KUKA KRL program: MyProgram_241().src

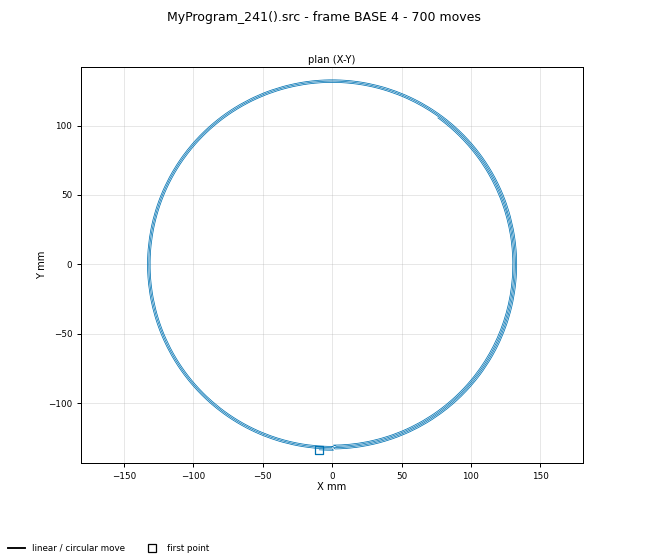
[picture p0: tool path of MyProgram_241().src in frame BASE 4, 700 of 700 moves have a stored position in this frame; points joined in program order, loops and branches not executed]
&ACCESS RVP
&REL 1
&PARAM TEMPLATE = C:\KRC\Roboter\Template\vorgabe
&PARAM EDITMASK = *
DEF MyProgram_241()
; ---- Setting reference (Base) ----
$BASE = BASE_DATA[4]

; --------------------------
; ---- Setting tool (TCP) ----
$TOOL = TOOL_DATA[3]
; --------------------------

$VEL.CP = VEL_APROX_PRINT
Startdeposition()
$VEL.CP = VEL_PRINT
LIN {X -9.2495,Y -133.5203,Z 161,A -94.9072,B 19.4805,C -0.419,E1 19.4752,E2 543.1799} C_DIS
LIN {X -6.5634,Y -133.6784,Z 161,A -93.7655,B 19.4805,C -0.4187,E1 19.4784,E2 542.039} C_DIS
LIN {X -3.4511,Y -133.7952,Z 161,A -92.3278,B 19.4805,C -0.4231,E1 19.4824,E2 540.5877} C_DIS
LIN {X 0.9612,Y -133.8342,Z 161,A -90.53,B 19.4805,C -0.4197,E1 19.4874,E2 538.8002} C_DIS
Enddeposition()
LIN {X 0.9612,Y -133.8342,Z 161,A -90.53,B 19.4805,C -0.4197,E1 19.4874,E2 538.8002} C_DIS
Startdeposition()
$VEL.CP = VEL_PRINT
LIN {X 0.1384,Y -132.9165,Z 161,A -91.2361,B 18.2986,C -0.2589,E1 18.2997,E2 539.9083} C_DIS
LIN {X -4.1167,Y -132.8521,Z 161,A -93.0475,B 18.2986,C -0.2596,E1 18.2947,E2 541.7178} C_DIS
LIN {X -8.2426,Y -132.6594,Z 161,A -94.8169,B 18.2986,C -0.26,E1 18.2897,E2 543.4865} C_DIS
LIN {X -12.4116,Y -132.3347,Z 161,A -96.6477,B 18.2986,C -0.2591,E1 18.2846,E2 545.3213} C_DIS
LIN {X -16.3847,Y -131.9029,Z 161,A -98.3665,B 18.2986,C -0.2596,E1 18.2799,E2 547.0403} C_DIS
LIN {X -20.2854,Y -131.3579,Z 161,A -99.987,B 18.2986,C -0.263,E1 18.2754,E2 548.6519} C_DIS
LIN {X -24.0292,Y -130.7264,Z 161,A -101.7483,B 18.2986,C -0.2589,E1 18.2705,E2 550.4286} C_DIS
LIN {X -28.0957,Y -129.9116,Z 161,A -103.4109,B 18.2986,C -0.2644,E1 18.266,E2 552.0765} C_DIS
LIN {X -35.5368,Y -128.0764,Z 161,A -106.7188,B 18.2985,C -0.2661,E1 18.2571,E2 555.3853} C_DIS
LIN {X -38.6101,Y -127.1837,Z 161,A -107.9788,B 18.2984,C -0.2716,E1 18.2537,E2 556.6309} C_DIS
LIN {X -43.386,Y -125.6345,Z 161,A -110.1035,B 18.2984,C -0.2748,E1 18.2481,E2 558.7509} C_DIS
LIN {X -46.3353,Y -124.5771,Z 161,A -111.6534,B 18.2984,C -0.2686,E1 18.244,E2 560.3249} C_DIS
LIN {X -49.0204,Y -123.547,Z 161,A -112.8623,B 18.2984,C -0.2709,E1 18.2408,E2 561.5301} C_DIS
LIN {X -52.3507,Y -122.1716,Z 161,A -114.4846,B 18.2984,C -0.27,E1 18.2366,E2 563.1605} C_DIS
LIN {X -55.4455,Y -120.7984,Z 161,A -115.9124,B 18.2984,C -0.2728,E1 18.233,E2 564.5843} C_DIS
LIN {X -58.5683,Y -119.3152,Z 161,A -117.3737,B 18.2984,C -0.2756,E1 18.2294,E2 566.0418} C_DIS
LIN {X -61.6117,Y -117.7724,Z 161,A -118.8799,B 18.2984,C -0.2762,E1 18.2256,E2 567.5519} C_DIS
LIN {X -65.3546,Y -115.7397,Z 161,A -120.716,B 18.2983,C -0.2786,E1 18.2211,E2 569.3877} C_DIS
LIN {X -68.6279,Y -113.8291,Z 161,A -122.4205,B 18.2983,C -0.2784,E1 18.217,E2 571.1001} C_DIS
LIN {X -72.315,Y -111.523,Z 161,A -124.324,B 18.2983,C -0.2802,E1 18.2125,E2 573.0064} C_DIS
LIN {X -75.3253,Y -109.5123,Z 161,A -126.0329,B 18.2983,C -0.2774,E1 18.2085,E2 574.7324} C_DIS
LIN {X -78.2414,Y -107.4486,Z 161,A -127.5386,B 18.2983,C -0.2812,E1 18.2051,E2 576.2334} C_DIS
LIN {X -82.235,Y -104.4235,Z 161,A -129.4084,B 18.298,C -0.2954,E1 18.2011,E2 578.0674} C_DIS
LIN {X -86.685,Y -100.7598,Z 161,A -132.0769,B 18.298,C -0.2934,E1 18.1953,E2 580.7566} C_DIS
LIN {X -90.3322,Y -97.504,Z 161,A -134.3348,B 18.298,C -0.2922,E1 18.1906,E2 583.0312} C_DIS
LIN {X -93.9479,Y -94.0253,Z 161,A -136.4373,B 18.298,C -0.2987,E1 18.1864,E2 585.1252} C_DIS
LIN {X -97.0592,Y -90.8099,Z 161,A -138.3595,B 18.298,C -0.3031,E1 18.1827,E2 587.0452} C_DIS
LIN {X -101.3952,Y -85.9412,Z 161,A -141.1571,B 18.2978,C -0.3098,E1 18.1776,E2 589.8391} C_DIS
LIN {X -103.6083,Y -83.2598,Z 161,A -142.773,B 18.2978,C -0.3091,E1 18.1747,E2 591.4678} C_DIS
LIN {X -106.4807,Y -79.5533,Z 161,A -144.7225,B 18.2978,C -0.3164,E1 18.1714,E2 593.407} C_DIS
LIN {X -109.0968,Y -75.9258,Z 161,A -146.6648,B 18.2976,C -0.3206,E1 18.1683,E2 595.3493} C_DIS
LIN {X -110.9412,Y -73.2045,Z 161,A -147.9595,B 18.2975,C -0.3284,E1 18.1663,E2 596.628} C_DIS
LIN {X -113.1832,Y -69.6881,Z 161,A -149.914,B 18.2975,C -0.3275,E1 18.1634,E2 598.5995} C_DIS
LIN {X -115.5866,Y -65.625,Z 161,A -151.9354,B 18.2975,C -0.3332,E1 18.1606,E2 600.6173} C_DIS
LIN {X -117.4844,Y -62.1602,Z 161,A -153.6006,B 18.2973,C -0.3391,E1 18.1584,E2 602.2761} C_DIS
LIN {X -118.8433,Y -59.525,Z 161,A -155.4953,B 18.2976,C -0.3212,E1 18.1559,E2 604.2426} C_DIS
LIN {X -120.9937,Y -55.0223,Z 161,A -157.1772,B 18.2972,C -0.3432,E1 18.154,E2 605.8667} C_DIS
LIN {X -122.5718,Y -51.4053,Z 161,A -158.7371,B 18.2971,C -0.3529,E1 18.1523,E2 607.4078} C_DIS
LIN {X -124.1426,Y -47.4915,Z 161,A -160.6737,B 18.2971,C -0.3539,E1 18.1503,E2 609.3565} C_DIS
LIN {X -125.4984,Y -43.7786,Z 161,A -162.2899,B 18.2969,C -0.3618,E1 18.1488,E2 610.9603} C_DIS
LIN {X -126.4864,Y -40.8374,Z 161,A -163.639,B 18.2969,C -0.3653,E1 18.1476,E2 612.3091} C_DIS
LIN {X -127.5295,Y -37.4513,Z 161,A -165.1262,B 18.2967,C -0.3712,E1 18.1464,E2 613.7896} C_DIS
LIN {X -128.4618,Y -34.1165,Z 161,A -166.6183,B 18.2967,C -0.3756,E1 18.1453,E2 615.2798} C_DIS
LIN {X -129.2371,Y -31.0509,Z 161,A -168.1072,B 18.2967,C -0.3753,E1 18.1443,E2 616.7819} C_DIS
LIN {X -130.3279,Y -26.0999,Z 161,A -170.7821,B 18.2968,C -0.3652,E1 18.1428,E2 619.5116} C_DIS
LIN {X -131.1102,Y -21.829,Z 161,A -172.1204,B 18.2964,C -0.389,E1 18.1422,E2 620.7845} C_DIS
LIN {X -132.1507,Y -14.2347,Z 161,A -175.3713,B 18.2961,C -0.4009,E1 18.141,E2 624.0247} C_DIS
LIN {X -132.5626,Y -9.6743,Z 161,A -177.4773,B 18.2961,C -0.4024,E1 18.1405,E2 626.1437} C_DIS
LIN {X -132.7947,Y -5.6803,Z 161,A -179.2819,B 18.2961,C -0.405,E1 18.1402,E2 627.9553} C_DIS
LIN {X -132.8975,Y -2.1736,Z 161,A 179.0637,B 18.2961,C -0.4049,E1 18.1402,E2 629.6243} C_DIS
LIN {X -132.8525,Y 4.1024,Z 161,A 176.4408,B 18.2958,C -0.4161,E1 18.1402,E2 632.2336} C_DIS
LIN {X -132.6983,Y 7.6106,Z 161,A 175.0478,B 18.2956,C -0.4249,E1 18.1405,E2 633.6102} C_DIS
LIN {X -132.4708,Y 10.8636,Z 161,A 173.4125,B 18.2956,C -0.4214,E1 18.1408,E2 635.2704} C_DIS
LIN {X -131.5776,Y 18.8081,Z 161,A 170.1547,B 18.2953,C -0.4385,E1 18.1419,E2 638.5009} C_DIS
LIN {X -130.5143,Y 25.1485,Z 161,A 167.5088,B 18.295,C -0.4513,E1 18.1431,E2 641.1279} C_DIS
LIN {X -129.9099,Y 28.1034,Z 161,A 165.8704,B 18.2951,C -0.4437,E1 18.1441,E2 642.8043} C_DIS
LIN {X -128.9068,Y 32.3961,Z 161,A 164.0424,B 18.295,C -0.452,E1 18.1453,E2 644.6209} C_DIS
LIN {X -127.9085,Y 36.1373,Z 161,A 162.5056,B 18.2947,C -0.4615,E1 18.1464,E2 646.1395} C_DIS
LIN {X -127.1123,Y 38.8434,Z 161,A 161.1487,B 18.2947,C -0.4604,E1 18.1475,E2 647.5111} C_DIS
LIN {X -125.9761,Y 42.3856,Z 161,A 159.4471,B 18.2947,C -0.4618,E1 18.149,E2 649.222} C_DIS
LIN {X -124.5771,Y 46.3353,Z 161,A 157.7541,B 18.2945,C -0.4711,E1 18.1506,E2 650.8988} C_DIS
LIN {X -123.4617,Y 49.2319,Z 161,A 156.3149,B 18.2945,C -0.4715,E1 18.1521,E2 652.3479} C_DIS
LIN {X -121.7094,Y 53.4197,Z 161,A 154.3178,B 18.2944,C -0.4758,E1 18.1543,E2 654.3468} C_DIS
LIN {X -120.3554,Y 56.4034,Z 161,A 152.712,B 18.2944,C -0.4733,E1 18.1562,E2 655.9732} C_DIS
LIN {X -117.2326,Y 62.6373,Z 161,A 149.8455,B 18.2941,C -0.4865,E1 18.1598,E2 658.8189} C_DIS
LIN {X -115.0744,Y 66.5186,Z 161,A 147.9625,B 18.2939,C -0.4929,E1 18.1624,E2 660.6954} C_DIS
LIN {X -111.8673,Y 71.7814,Z 161,A 145.5439,B 18.2935,C -0.5083,E1 18.1659,E2 663.082} C_DIS
LIN {X -109.3103,Y 75.619,Z 161,A 143.2666,B 18.2937,C -0.5035,E1 18.1695,E2 665.3906} C_DIS
LIN {X -107.5089,Y 78.1583,Z 161,A 141.7554,B 18.2937,C -0.5012,E1 18.172,E2 666.9196} C_DIS
LIN {X -104.4685,Y 82.1776,Z 161,A 139.7656,B 18.2934,C -0.513,E1 18.1753,E2 668.8849} C_DIS
LIN {X -101.1528,Y 86.2263,Z 161,A 137.4556,B 18.2933,C -0.5167,E1 18.1795,E2 671.1981} C_DIS
LIN {X -98.371,Y 89.3867,Z 161,A 135.1653,B 18.2936,C -0.5046,E1 18.1838,E2 673.5414} C_DIS
LIN {X -95.2866,Y 92.6682,Z 161,A 133.1063,B 18.2936,C -0.5051,E1 18.1879,E2 675.6114} C_DIS
LIN {X -91.7254,Y 96.1941,Z 161,A 131.4773,B 18.293,C -0.5283,E1 18.191,E2 677.1755} C_DIS
LIN {X -88.6456,Y 99.0393,Z 161,A 129.1931,B 18.2933,C -0.5157,E1 18.1959,E2 679.5131} C_DIS
LIN {X -85.1654,Y 102.0472,Z 161,A 127.6555,B 18.2928,C -0.5353,E1 18.199,E2 680.9961} C_DIS
LIN {X -81.5235,Y 104.9798,Z 161,A 125.6332,B 18.2927,C -0.5392,E1 18.2035,E2 683.0166} C_DIS
LIN {X -79.1259,Y 106.799,Z 161,A 124.0795,B 18.2929,C -0.5327,E1 18.207,E2 684.5987} C_DIS
LIN {X -76.2561,Y 108.8669,Z 161,A 122.7949,B 18.2925,C -0.544,E1 18.2099,E2 685.8534} C_DIS
LIN {X -72.7549,Y 111.2372,Z 161,A 120.7525,B 18.2927,C -0.5396,E1 18.2147,E2 687.9194} C_DIS
LIN {X -69.9728,Y 113.0077,Z 161,A 119.5284,B 18.2924,C -0.5491,E1 18.2175,E2 689.1187} C_DIS
LIN {X -66.1509,Y 115.2866,Z 161,A 117.5766,B 18.2924,C -0.5511,E1 18.2222,E2 691.0723} C_DIS
LIN {X -58.8014,Y 119.2003,Z 161,A 114.419,B 18.2917,C -0.5721,E1 18.2299,E2 694.1751} C_DIS
LIN {X -56.2098,Y 120.445,Z 161,A 112.8618,B 18.292,C -0.5625,E1 18.2339,E2 695.7685} C_DIS
LIN {X -50.1924,Y 123.0745,Z 161,A 110.0183,B 18.2919,C -0.5658,E1 18.2412,E2 698.6107} C_DIS
LIN {X -46.8336,Y 124.3905,Z 161,A 108.4481,B 18.2919,C -0.5672,E1 18.2453,E2 700.1811} C_DIS
LIN {X -43.5527,Y 125.5767,Z 161,A 107.165,B 18.2916,C -0.5769,E1 18.2486,E2 701.4368} C_DIS
LIN {X -35.6772,Y 128.0371,Z 161,A 103.34,B 18.2917,C -0.5708,E1 18.2589,E2 705.2905} C_DIS
LIN {X -32.6139,Y 128.8515,Z 161,A 101.1386,B 18.2926,C -0.542,E1 18.2651,E2 707.5883} C_DIS
LIN {X -26.5557,Y 130.2351,Z 161,A 99.351,B 18.2916,C -0.5762,E1 18.2697,E2 709.2698} C_DIS
LIN {X -21.364,Y 131.1878,Z 161,A 96.9781,B 18.2916,C -0.5741,E1 18.2763,E2 711.6525} C_DIS
LIN {X -18.0851,Y 131.6809,Z 161,A 95.4746,B 18.2917,C -0.5722,E1 18.2804,E2 713.1639} C_DIS
LIN {X -14.1509,Y 132.1597,Z 161,A 93.8546,B 18.2916,C -0.5763,E1 18.2849,E2 714.7723} C_DIS
LIN {X -9.6018,Y 132.5679,Z 161,A 91.9426,B 18.2915,C -0.5791,E1 18.2902,E2 716.6764} C_DIS
LIN {X -5.6691,Y 132.7951,Z 161,A 90.1665,B 18.2915,C -0.5767,E1 18.2952,E2 718.4609} C_DIS
LIN {X -1.9946,Y 132.9004,Z 161,A 88.5541,B 18.2915,C -0.576,E1 18.2997,E2 720.0756} C_DIS
LIN {X 2.2636,Y 132.896,Z 161,A 86.7933,B 18.2915,C -0.579,E1 18.3046,E2 721.8267} C_DIS
LIN {X 6.1173,Y 132.7755,Z 161,A 85.073,B 18.2915,C -0.5768,E1 18.3094,E2 723.5533} C_DIS
LIN {X 9.8935,Y 132.5466,Z 161,A 83.4557,B 18.2915,C -0.5772,E1 18.3139,E2 725.1683} C_DIS
LIN {X 13.9585,Y 132.1804,Z 161,A 81.7642,B 18.2915,C -0.5794,E1 18.3186,E2 726.8512} C_DIS
LIN {X 17.9465,Y 131.6997,Z 161,A 79.9117,B 18.2916,C -0.5744,E1 18.3237,E2 728.7175} C_DIS
LIN {X 21.8698,Y 131.1034,Z 161,A 78.308,B 18.2916,C -0.5778,E1 18.3281,E2 730.308} C_DIS
LIN {X 25.9086,Y 130.3668,Z 161,A 76.647,B 18.2914,C -0.5811,E1 18.3326,E2 731.9558} C_DIS
LIN {X 32.5426,Y 128.8696,Z 161,A 73.6385,B 18.2916,C -0.5765,E1 18.3409,E2 734.9731} C_DIS
LIN {X 36.3116,Y 127.8597,Z 161,A 71.5304,B 18.2921,C -0.5592,E1 18.3467,E2 737.1315} C_DIS
LIN {X 39.9998,Y 126.754,Z 161,A 70.3305,B 18.2916,C -0.5753,E1 18.3497,E2 738.2769} C_DIS
LIN {X 43.0105,Y 125.7647,Z 161,A 68.9706,B 18.2916,C -0.5744,E1 18.3533,E2 739.636} C_DIS
LIN {X 45.9963,Y 124.7041,Z 161,A 67.5722,B 18.2917,C -0.5719,E1 18.357,E2 741.0385} C_DIS
LIN {X 49.2285,Y 123.4631,Z 161,A 66.0066,B 18.2918,C -0.5676,E1 18.3611,E2 742.6128} C_DIS
LIN {X 52.1354,Y 122.2647,Z 161,A 64.6266,B 18.2919,C -0.5651,E1 18.3646,E2 743.9959} C_DIS
LIN {X 55.6121,Y 120.7214,Z 161,A 63.1407,B 18.2918,C -0.5692,E1 18.3684,E2 745.4637} C_DIS
LIN {X 58.4638,Y 119.3668,Z 161,A 61.659,B 18.292,C -0.5628,E1 18.3721,E2 746.9601} C_DIS
LIN {X 61.5588,Y 117.8002,Z 161,A 60.3125,B 18.2919,C -0.5667,E1 18.3754,E2 748.2891} C_DIS
LIN {X 64.8395,Y 116.0292,Z 161,A 58.3593,B 18.2923,C -0.551,E1 18.3803,E2 750.284} C_DIS
LIN {X 69.7639,Y 113.1368,Z 161,A 56.1128,B 18.2922,C -0.5557,E1 18.3856,E2 752.5057} C_DIS
LIN {X 72.5388,Y 111.3777,Z 161,A 54.5813,B 18.2924,C -0.549,E1 18.3893,E2 754.0514} C_DIS
LIN {X 76.5622,Y 108.6511,Z 161,A 52.6527,B 18.2924,C -0.552,E1 18.3937,E2 755.9612} C_DIS
LIN {X 79.5439,Y 106.4878,Z 161,A 51.0769,B 18.2924,C -0.5498,E1 18.3972,E2 757.5362} C_DIS
LIN {X 82.9963,Y 103.8196,Z 161,A 49.1969,B 18.2924,C -0.5464,E1 18.4013,E2 759.417} C_DIS
LIN {X 86.2012,Y 101.1741,Z 161,A 47.6289,B 18.2924,C -0.5518,E1 18.4046,E2 760.9592} C_DIS
LIN {X 88.4858,Y 99.1825,Z 161,A 46.0667,B 18.2927,C -0.5392,E1 18.408,E2 762.5529} C_DIS
LIN {X 91.638,Y 96.2776,Z 161,A 44.206,B 18.2927,C -0.5349,E1 18.4118,E2 764.4163} C_DIS
LIN {X 94.7689,Y 93.1972,Z 161,A 42.3316,B 18.2929,C -0.5317,E1 18.4155,E2 766.2897} C_DIS
LIN {X 97.8846,Y 89.919,Z 161,A 40.4415,B 18.2929,C -0.5298,E1 18.4191,E2 768.174} C_DIS
LIN {X 100.7888,Y 86.6514,Z 161,A 38.5452,B 18.2931,C -0.5251,E1 18.4226,E2 770.0733} C_DIS
LIN {X 103.5479,Y 83.3348,Z 161,A 36.7171,B 18.2931,C -0.5221,E1 18.4258,E2 771.8991} C_DIS
LIN {X 106.3042,Y 79.7895,Z 161,A 35.0309,B 18.2931,C -0.5275,E1 18.4286,E2 773.5569} C_DIS
LIN {X 108.3782,Y 76.9491,Z 161,A 33.2546,B 18.2934,C -0.5133,E1 18.4316,E2 775.3658} C_DIS
LIN {X 110.7131,Y 73.5495,Z 161,A 31.5005,B 18.2934,C -0.5099,E1 18.4343,E2 777.1187} C_DIS
LIN {X 113.0864,Y 69.846,Z 161,A 29.5766,B 18.2936,C -0.5039,E1 18.4372,E2 779.0478} C_DIS
LIN {X 115.2984,Y 66.1302,Z 161,A 27.7488,B 18.2937,C -0.5005,E1 18.4397,E2 780.8731} C_DIS
LIN {X 117.2716,Y 62.5648,Z 161,A 26.1184,B 18.2937,C -0.5009,E1 18.4419,E2 782.4901} C_DIS
LIN {X 119.568,Y 58.0493,Z 161,A 23.7869,B 18.294,C -0.4891,E1 18.4448,E2 784.8416} C_DIS
LIN {X 121.423,Y 54.063,Z 161,A 22.0564,B 18.294,C -0.4905,E1 18.4468,E2 786.5544} C_DIS
LIN {X 123.0251,Y 50.3149,Z 161,A 20.3228,B 18.294,C -0.4865,E1 18.4487,E2 788.2873} C_DIS
LIN {X 124.4107,Y 46.7796,Z 161,A 18.7119,B 18.2942,C -0.4829,E1 18.4503,E2 789.8968} C_DIS
LIN {X 125.4984,Y 43.7786,Z 161,A 16.3718,B 18.2952,C -0.44,E1 18.4526,E2 792.354} C_DIS
LIN {X 127.5601,Y 37.3467,Z 161,A 14.5164,B 18.2944,C -0.4742,E1 18.454,E2 794.0866} C_DIS
LIN {X 128.4063,Y 34.3248,Z 161,A 13.178,B 18.2944,C -0.4707,E1 18.4549,E2 795.425} C_DIS
LIN {X 130.4362,Y 25.557,Z 161,A 9.1636,B 18.2949,C -0.4535,E1 18.4574,E2 799.4609} C_DIS
LIN {X 131.0985,Y 21.8993,Z 161,A 7.6439,B 18.2949,C -0.4521,E1 18.4581,E2 800.9727} C_DIS
LIN {X 131.733,Y 17.6921,Z 161,A 5.8,B 18.2951,C -0.4461,E1 18.4589,E2 802.8203} C_DIS
LIN {X 132.1524,Y 14.2184,Z 161,A 4.3647,B 18.2951,C -0.4444,E1 18.4593,E2 804.2489} C_DIS
LIN {X 132.5024,Y 10.4902,Z 161,A 2.6196,B 18.2954,C -0.4341,E1 18.4597,E2 806.0121} C_DIS
LIN {X 132.753,Y 6.5658,Z 161,A 1.0613,B 18.2954,C -0.4345,E1 18.46,E2 807.5562} C_DIS
LIN {X 132.8946,Y 2.3468,Z 161,A -0.7456,B 18.2954,C -0.4293,E1 18.4601,E2 809.3641} C_DIS
LIN {X 132.903,Y -1.8399,Z 161,A -2.5484,B 18.2956,C -0.4238,E1 18.4601,E2 811.1693} C_DIS
LIN {X 132.7988,Y -5.5747,Z 161,A -4.165,B 18.2957,C -0.4186,E1 18.4599,E2 812.789} C_DIS
LIN {X 132.582,Y -9.4089,Z 161,A -5.6521,B 18.2957,C -0.4203,E1 18.4597,E2 814.2581} C_DIS
LIN {X 132.3045,Y -12.7262,Z 161,A -7.1824,B 18.2959,C -0.4119,E1 18.4593,E2 815.8021} C_DIS
LIN {X 131.8591,Y -16.7295,Z 161,A -8.9297,B 18.2959,C -0.4061,E1 18.4587,E2 817.5534} C_DIS
LIN {X 131.3852,Y -20.1091,Z 161,A -10.261,B 18.2959,C -0.4073,E1 18.4582,E2 818.8698} C_DIS
LIN {X 130.707,Y -24.1373,Z 161,A -12.0743,B 18.2961,C -0.3997,E1 18.4573,E2 820.6923} C_DIS
LIN {X 130.2581,Y -26.4425,Z 161,A -13.5134,B 18.2966,C -0.3791,E1 18.4565,E2 822.1845} C_DIS
LIN {X 129.4057,Y -30.3501,Z 161,A -14.9445,B 18.2964,C -0.3858,E1 18.4556,E2 823.5829} C_DIS
LIN {X 128.4854,Y -34.0282,Z 161,A -16.5267,B 18.2964,C -0.383,E1 18.4545,E2 825.1612} C_DIS
LIN {X 126.8516,Y -39.6943,Z 161,A -19.0884,B 18.2966,C -0.3744,E1 18.4525,E2 827.7292} C_DIS
LIN {X 125.8144,Y -42.867,Z 161,A -20.4323,B 18.2966,C -0.374,E1 18.4513,E2 829.0638} C_DIS
LIN {X 123.5893,Y -48.915,Z 161,A -23.1404,B 18.2968,C -0.3686,E1 18.4487,E2 831.7677} C_DIS
LIN {X 122.1903,Y -52.3074,Z 161,A -24.76,B 18.2968,C -0.3625,E1 18.4469,E2 833.3942} C_DIS
LIN {X 120.9323,Y -55.1559,Z 161,A -26.0199,B 18.2968,C -0.3619,E1 18.4454,E2 834.6462} C_DIS
LIN {X 119.8223,Y -57.5238,Z 161,A -27.5375,B 18.2972,C -0.3428,E1 18.4436,E2 836.2128} C_DIS
LIN {X 118.11,Y -60.9663,Z 161,A -28.788,B 18.297,C -0.3546,E1 18.442,E2 837.4166} C_DIS
LIN {X 115.5802,Y -65.6363,Z 161,A -31.1832,B 18.2972,C -0.3439,E1 18.4388,E2 839.828} C_DIS
LIN {X 113.2454,Y -69.5867,Z 161,A -33.101,B 18.2972,C -0.3409,E1 18.436,E2 841.7415} C_DIS
LIN {X 108.6446,Y -76.5715,Z 161,A -36.6755,B 18.2974,C -0.3325,E1 18.4305,E2 845.3176} C_DIS
LIN {X 106.832,Y -79.0816,Z 161,A -38.5852,B 18.2979,C -0.3058,E1 18.4272,E2 847.2989} C_DIS
LIN {X 103.7123,Y -83.1309,Z 161,A -40.1691,B 18.2976,C -0.3252,E1 18.4246,E2 848.811} C_DIS
LIN {X 99.3901,Y -88.2526,Z 161,A -43.0913,B 18.2976,C -0.3167,E1 18.4192,E2 851.7414} C_DIS
LIN {X 96.4836,Y -91.4212,Z 161,A -44.8791,B 18.2977,C -0.3149,E1 18.4158,E2 853.5238} C_DIS
LIN {X 92.8693,Y -95.0905,Z 161,A -47.4879,B 18.2981,C -0.2941,E1 18.4106,E2 856.1828} C_DIS
LIN {X 89.939,Y -97.8663,Z 161,A -48.8311,B 18.2979,C -0.3062,E1 18.4079,E2 857.4802} C_DIS
LIN {X 86.6185,Y -100.8171,Z 161,A -50.759,B 18.2979,C -0.3015,E1 18.4038,E2 859.4122} C_DIS
LIN {X 82.5695,Y -104.1592,Z 161,A -53.6206,B 18.2984,C -0.2729,E1 18.3975,E2 862.3492} C_DIS
LIN {X 78.2861,Y -107.4162,Z 161,A -55.1166,B 18.298,C -0.3011,E1 18.3943,E2 863.7483} C_DIS
LIN {X 72.067,Y -111.684,Z 161,A -58.5768,B 18.2982,C -0.2866,E1 18.3863,E2 867.238} C_DIS
LIN {X 68.2867,Y -114.0343,Z 161,A -60.4894,B 18.2982,C -0.2834,E1 18.3817,E2 869.1521} C_DIS
LIN {X 61.9747,Y -117.5818,Z 161,A -63.5046,B 18.2982,C -0.2825,E1 18.3744,E2 872.1579} C_DIS
LIN {X 56.076,Y -120.5068,Z 161,A -66.2112,B 18.2982,C -0.2834,E1 18.3676,E2 874.8515} C_DIS
LIN {X 52.9845,Y -121.8976,Z 161,A -67.6936,B 18.2982,C -0.2804,E1 18.3638,E2 876.3381} C_DIS
LIN {X 49.9471,Y -123.1734,Z 161,A -69.0655,B 18.2982,C -0.2804,E1 18.3603,E2 877.7055} C_DIS
LIN {X 47.0695,Y -124.3021,Z 161,A -70.5604,B 18.2984,C -0.2723,E1 18.3563,E2 879.2215} C_DIS
LIN {X 43.2872,Y -125.6687,Z 161,A -72.906,B 18.2987,C -0.2464,E1 18.3499,E2 881.6427} C_DIS
LIN {X 38.2313,Y -127.2997,Z 161,A -74.6409,B 18.2985,C -0.2655,E1 18.3455,E2 883.3128} C_DIS
LIN {X 34.0095,Y -128.4904,Z 161,A -76.4951,B 18.2985,C -0.265,E1 18.3405,E2 885.1641} C_DIS
LIN {X 29.8513,Y -129.5197,Z 161,A -78.2062,B 18.2985,C -0.2686,E1 18.3359,E2 886.8601} C_DIS
LIN {X 24.9022,Y -130.5614,Z 161,A -80.4336,B 18.2985,C -0.2651,E1 18.3298,E2 889.095} C_DIS
LIN {X 20.8815,Y -131.2656,Z 161,A -82.2608,B 18.2985,C -0.2612,E1 18.3247,E2 890.9318} C_DIS
LIN {X 17.3629,Y -131.7761,Z 161,A -83.6828,B 18.2985,C -0.2646,E1 18.3208,E2 892.3413} C_DIS
LIN {X 13.509,Y -132.2287,Z 161,A -85.5097,B 18.2985,C -0.2578,E1 18.3157,E2 894.1881} C_DIS
LIN {X 9.7818,Y -132.5548,Z 161,A -86.8692,B 18.2985,C -0.2668,E1 18.312,E2 895.5178} C_DIS
LIN {X 6.2095,Y -132.7709,Z 161,A -88.6098,B 18.2985,C -0.2587,E1 18.3071,E2 897.2833} C_DIS
LIN {X 2.1696,Y -132.8975,Z 161,A -90.2939,B 18.2985,C -0.2605,E1 18.3024,E2 898.9613} C_DIS
LIN {X 2.1696,Y -132.8975,Z 161,A -90.2939,B 18.2985,C -0.2605,E1 18.3024,E2 898.9613} C_DIS
Enddeposition()
LIN {X 0.9405,Y -131.9868,Z 161,A -89.6882,B 16.7079,C -0.1256,E1 16.7111,E2 898.6993} C_DIS
Startdeposition()
$VEL.CP = VEL_PRINT
LIN {X 4.7448,Y -131.9063,Z 161,A -87.9777,B 16.7079,C -0.128,E1 16.7159,E2 896.9809} C_DIS
LIN {X 8.297,Y -131.7301,Z 161,A -86.442,B 16.7079,C -0.1283,E1 16.7202,E2 895.4453} C_DIS
LIN {X 12.5703,Y -131.391,Z 161,A -84.6053,B 16.7079,C -0.1283,E1 16.7253,E2 893.6104} C_DIS
LIN {X 16.3347,Y -130.9781,Z 161,A -82.8484,B 16.7079,C -0.1331,E1 16.7302,E2 891.8387} C_DIS
LIN {X 20.0531,Y -130.4587,Z 161,A -81.3784,B 16.7079,C -0.1284,E1 16.7342,E2 890.387} C_DIS
LIN {X 23.0656,Y -129.9599,Z 161,A -80.0042,B 16.7079,C -0.131,E1 16.738,E2 889.0059} C_DIS
LIN {X 25.9574,Y -129.4137,Z 161,A -78.8482,B 16.7079,C -0.1277,E1 16.7411,E2 887.8638} C_DIS
LIN {X 29.6579,Y -128.6158,Z 161,A -77.0787,B 16.7079,C -0.1335,E1 16.746,E2 886.0776} C_DIS
LIN {X 34.0718,Y -127.5173,Z 161,A -75.2068,B 16.7079,C -0.1317,E1 16.751,E2 884.2167} C_DIS
LIN {X 37.2508,Y -126.6252,Z 161,A -73.4085,B 16.7078,C -0.1463,E1 16.756,E2 882.3725} C_DIS
LIN {X 40.3687,Y -125.666,Z 161,A -72.0648,B 16.7078,C -0.1452,E1 16.7595,E2 881.0365} C_DIS
LIN {X 44.2514,Y -124.3528,Z 161,A -70.4396,B 16.7078,C -0.1417,E1 16.7638,E2 879.4285} C_DIS
LIN {X 47.654,Y -123.0879,Z 161,A -68.9392,B 16.7078,C -0.1409,E1 16.7677,E2 877.9358} C_DIS
LIN {X 51.148,Y -121.6777,Z 161,A -67.2567,B 16.7078,C -0.1448,E1 16.772,E2 876.246} C_DIS
LIN {X 55.4496,Y -119.7782,Z 161,A -64.7385,B 16.7076,C -0.1651,E1 16.7786,E2 873.6672} C_DIS
LIN {X 59.5929,Y -117.7721,Z 161,A -63.2907,B 16.7078,C -0.148,E1 16.782,E2 872.285} C_DIS
LIN {X 65.3843,Y -114.6599,Z 161,A -60.4782,B 16.7078,C -0.151,E1 16.7889,E2 869.4746} C_DIS
LIN {X 68.6356,Y -112.7445,Z 161,A -58.7572,B 16.7077,C -0.1569,E1 16.7931,E2 867.7417} C_DIS
LIN {X 71.1136,Y -111.1974,Z 161,A -56.6149,B 16.7073,C -0.1916,E1 16.7984,E2 865.4901} C_DIS
LIN {X 76.6558,Y -107.4519,Z 161,A -54.6011,B 16.7076,C -0.1639,E1 16.8027,E2 863.5828} C_DIS
LIN {X 80.1974,Y -104.835,Z 161,A -52.4802,B 16.7076,C -0.1755,E1 16.8075,E2 861.434} C_DIS
LIN {X 82.7891,Y -102.8007,Z 161,A -51.6072,B 16.7076,C -0.1577,E1 16.8093,E2 860.6274} C_DIS
LIN {X 87.0427,Y -99.2255,Z 161,A -48.8617,B 16.7076,C -0.1751,E1 16.8152,E2 857.8382} C_DIS
LIN {X 92.9452,Y -93.7188,Z 161,A -45.5741,B 16.7076,C -0.1748,E1 16.8218,E2 854.5728} C_DIS
LIN {X 97.2491,Y -89.2448,Z 161,A -42.8013,B 16.7074,C -0.184,E1 16.8272,E2 851.787} C_DIS
LIN {X 101.6682,Y -84.1758,Z 161,A -39.8876,B 16.7074,C -0.1908,E1 16.8325,E2 848.8702} C_DIS
LIN {X 106.0715,Y -78.5554,Z 161,A -36.7827,B 16.7073,C -0.1988,E1 16.8378,E2 845.7605} C_DIS
LIN {X 108.2212,Y -75.566,Z 161,A -34.5716,B 16.7069,C -0.2261,E1 16.8415,E2 843.4718} C_DIS
LIN {X 111.1369,Y -71.2081,Z 161,A -32.9018,B 16.7071,C -0.2092,E1 16.8439,E2 841.8735} C_DIS
LIN {X 113.5575,Y -67.2816,Z 161,A -30.9195,B 16.7071,C -0.2139,E1 16.8467,E2 839.8908} C_DIS
LIN {X 115.1294,Y -64.5541,Z 161,A -29.2775,B 16.7069,C -0.228,E1 16.849,E2 838.2131} C_DIS
LIN {X 116.8044,Y -61.4673,Z 161,A -28.184,B 16.707,C -0.216,E1 16.8504,E2 837.1701} C_DIS
LIN {X 118.0417,Y -59.0609,Z 161,A -27.0184,B 16.707,C -0.2189,E1 16.8519,E2 836.0041} C_DIS
LIN {X 119.5185,Y -56.0113,Z 161,A -25.4954,B 16.707,C -0.225,E1 16.8537,E2 834.4726} C_DIS
LIN {X 120.9607,Y -52.8226,Z 161,A -23.9635,B 16.7069,C -0.2299,E1 16.8554,E2 832.9369} C_DIS
LIN {X 122.4371,Y -49.3017,Z 161,A -22.0997,B 16.7067,C -0.2425,E1 16.8574,E2 831.0454} C_DIS
LIN {X 124.498,Y -43.8425,Z 161,A -19.7319,B 16.7067,C -0.2436,E1 16.8597,E2 828.6943} C_DIS
LIN {X 125.6673,Y -40.3645,Z 161,A -18.2849,B 16.7067,C -0.2428,E1 16.8609,E2 827.2628} C_DIS
LIN {X 126.4998,Y -37.6792,Z 161,A -16.8861,B 16.7065,C -0.2532,E1 16.8621,E2 825.8405} C_DIS
LIN {X 127.8345,Y -32.8639,Z 161,A -14.9517,B 16.7065,C -0.2508,E1 16.8634,E2 823.9316} C_DIS
LIN {X 129.4384,Y -25.8362,Z 161,A -11.8414,B 16.7065,C -0.2595,E1 16.8653,E2 820.8194} C_DIS
LIN {X 130.1664,Y -21.8701,Z 161,A -10.0222,B 16.7063,C -0.2675,E1 16.8662,E2 818.9893} C_DIS
LIN {X 130.8014,Y -17.688,Z 161,A -8.2085,B 16.7063,C -0.2722,E1 16.8669,E2 817.1758} C_DIS
LIN {X 131.258,Y -13.8916,Z 161,A -6.5823,B 16.7062,C -0.276,E1 16.8674,E2 815.5513} C_DIS
LIN {X 131.6274,Y -9.7918,Z 161,A -4.8129,B 16.7062,C -0.2808,E1 16.8678,E2 813.7816} C_DIS
LIN {X 131.8688,Y -5.7073,Z 161,A -3.1521,B 16.7061,C -0.2819,E1 16.8681,E2 812.1324} C_DIS
LIN {X 131.9703,Y -2.3464,Z 161,A -1.6875,B 16.7061,C -0.2866,E1 16.8681,E2 810.6652} C_DIS
LIN {X 131.9872,Y 1.1315,Z 161,A -0.0209,B 16.7058,C -0.2971,E1 16.8681,E2 808.9775} C_DIS
LIN {X 131.9063,Y 4.7448,Z 161,A 1.4393,B 16.7058,C -0.2978,E1 16.8681,E2 807.5285} C_DIS
LIN {X 131.6984,Y 8.8115,Z 161,A 3.2077,B 16.7058,C -0.3032,E1 16.8678,E2 805.7577} C_DIS
LIN {X 131.4043,Y 12.4312,Z 161,A 4.7163,B 16.7057,C -0.3055,E1 16.8674,E2 804.2552} C_DIS
LIN {X 131.0322,Y 15.8814,Z 161,A 6.2136,B 16.7057,C -0.3097,E1 16.8669,E2 802.7571} C_DIS
LIN {X 130.4735,Y 19.9573,Z 161,A 7.9912,B 16.7055,C -0.3147,E1 16.8662,E2 800.9782} C_DIS
LIN {X 129.9128,Y 23.3292,Z 161,A 9.3328,B 16.7055,C -0.3138,E1 16.8656,E2 799.652} C_DIS
LIN {X 129.375,Y 26.1474,Z 161,A 11.729,B 16.7046,C -0.3613,E1 16.8642,E2 797.1138} C_DIS
LIN {X 127.7431,Y 33.2244,Z 161,A 13.926,B 16.7052,C -0.3341,E1 16.8627,E2 795.0301} C_DIS
LIN {X 124.6346,Y 43.4487,Z 161,A 18.3993,B 16.705,C -0.3412,E1 16.859,E2 790.5718} C_DIS
LIN {X 123.2718,Y 47.1811,Z 161,A 20.2417,B 16.7048,C -0.3504,E1 16.8572,E2 788.7134} C_DIS
LIN {X 121.8345,Y 50.7727,Z 161,A 21.5779,B 16.705,C -0.3423,E1 16.8558,E2 787.4167} C_DIS
LIN {X 120.6516,Y 53.5243,Z 161,A 23.125,B 16.7047,C -0.3551,E1 16.8541,E2 785.8386} C_DIS
LIN {X 118.0581,Y 59.0277,Z 161,A 25.676,B 16.7047,C -0.3588,E1 16.851,E2 783.2959} C_DIS
LIN {X 116.496,Y 62.0545,Z 161,A 27.1774,B 16.7046,C -0.3636,E1 16.849,E2 781.7904} C_DIS
LIN {X 114.7143,Y 65.2891,Z 161,A 28.8407,B 16.7044,C -0.3701,E1 16.8467,E2 780.1183} C_DIS
LIN {X 112.4647,Y 69.092,Z 161,A 30.717,B 16.7044,C -0.3734,E1 16.844,E2 778.2452} C_DIS
LIN {X 110.0427,Y 72.8885,Z 161,A 32.6446,B 16.7043,C -0.3773,E1 16.8411,E2 776.3193} C_DIS
LIN {X 108.0224,Y 75.8502,Z 161,A 34.0716,B 16.7043,C -0.3763,E1 16.8389,E2 774.9065} C_DIS
LIN {X 105.6256,Y 79.1543,Z 161,A 35.9914,B 16.7041,C -0.386,E1 16.8357,E2 772.9676} C_DIS
LIN {X 102.9605,Y 82.5909,Z 161,A 37.8957,B 16.704,C -0.391,E1 16.8323,E2 771.0598} C_DIS
LIN {X 100.0255,Y 86.1215,Z 161,A 39.8025,B 16.704,C -0.3923,E1 16.8289,E2 769.162} C_DIS
LIN {X 97.1169,Y 89.3886,Z 161,A 41.6759,B 16.7039,C -0.3955,E1 16.8254,E2 767.2903} C_DIS
LIN {X 94.3219,Y 92.333,Z 161,A 43.4752,B 16.7037,C -0.4006,E1 16.8219,E2 765.4855} C_DIS
LIN {X 91.1272,Y 95.4874,Z 161,A 45.4007,B 16.7037,C -0.4038,E1 16.8181,E2 763.5617} C_DIS
LIN {X 87.8692,Y 98.494,Z 161,A 47.3088,B 16.7036,C -0.407,E1 16.8141,E2 761.6544} C_DIS
LIN {X 84.7148,Y 101.2197,Z 161,A 49.1212,B 16.7036,C -0.4105,E1 16.8103,E2 759.8408} C_DIS
LIN {X 81.2118,Y 104.0519,Z 161,A 51.0449,B 16.7034,C -0.4129,E1 16.8061,E2 757.92} C_DIS
LIN {X 77.8342,Y 106.602,Z 161,A 52.9136,B 16.7034,C -0.4172,E1 16.8019,E2 756.0468} C_DIS
LIN {X 74.2705,Y 109.1147,Z 161,A 54.6482,B 16.7034,C -0.4146,E1 16.7979,E2 754.3304} C_DIS
LIN {X 70.9805,Y 111.2826,Z 161,A 56.3769,B 16.7034,C -0.4179,E1 16.7939,E2 752.5989} C_DIS
LIN {X 68.4653,Y 112.8474,Z 161,A 58.0032,B 16.703,C -0.4321,E1 16.7899,E2 750.9316} C_DIS
LIN {X 65.4873,Y 114.6012,Z 161,A 59.1678,B 16.7032,C -0.4222,E1 16.7872,E2 749.8068} C_DIS
LIN {X 62.0709,Y 116.4874,Z 161,A 60.9976,B 16.703,C -0.4293,E1 16.7826,E2 747.9604} C_DIS
LIN {X 58.5811,Y 118.2784,Z 161,A 62.4971,B 16.7032,C -0.4243,E1 16.779,E2 746.4848} C_DIS
LIN {X 55.7809,Y 119.6251,Z 161,A 63.9215,B 16.7031,C -0.4286,E1 16.7753,E2 745.0511} C_DIS
LIN {X 52.74,Y 120.9965,Z 161,A 65.2453,B 16.7031,C -0.4258,E1 16.772,E2 743.742} C_DIS
LIN {X 49.95,Y 122.1758,Z 161,A 66.6376,B 16.7031,C -0.4299,E1 16.7684,E2 742.3405} C_DIS
LIN {X 46.6153,Y 123.4854,Z 161,A 68.1632,B 16.7031,C -0.4305,E1 16.7644,E2 740.8182} C_DIS
LIN {X 43.173,Y 124.7301,Z 161,A 69.7672,B 16.703,C -0.4324,E1 16.7602,E2 739.2125} C_DIS
LIN {X 39.6836,Y 125.8848,Z 161,A 71.3346,B 16.703,C -0.4328,E1 16.756,E2 737.6485} C_DIS
LIN {X 33.2093,Y 127.7469,Z 161,A 74.2477,B 16.703,C -0.4344,E1 16.7482,E2 734.7372} C_DIS
LIN {X 26.0731,Y 129.3902,Z 161,A 77.4651,B 16.7028,C -0.4375,E1 16.7394,E2 731.5159} C_DIS
LIN {X 21.9983,Y 130.145,Z 161,A 79.3365,B 16.7028,C -0.4408,E1 16.7343,E2 729.6363} C_DIS
LIN {X 17.5537,Y 130.819,Z 161,A 81.2487,B 16.7028,C -0.4401,E1 16.729,E2 727.7294} C_DIS
LIN {X 13.974,Y 131.2492,Z 161,A 82.7689,B 16.7028,C -0.4389,E1 16.7248,E2 726.215} C_DIS
LIN {X 9.8405,Y 131.6238,Z 161,A 84.5953,B 16.7028,C -0.44,E1 16.7197,E2 724.3863} C_DIS
LIN {X 6.1721,Y 131.8474,Z 161,A 86.2236,B 16.7028,C -0.4412,E1 16.7151,E2 722.7548} C_DIS
LIN {X 2.6411,Y 131.9654,Z 161,A 87.734,B 16.7028,C -0.4403,E1 16.7109,E2 721.2478} C_DIS
LIN {X -0.8712,Y 131.9883,Z 161,A 89.2753,B 16.7028,C -0.4407,E1 16.7066,E2 719.7053} C_DIS
LIN {X -5.0786,Y 131.8933,Z 161,A 91.066,B 16.7028,C -0.4391,E1 16.7016,E2 717.9198} C_DIS
LIN {X -8.9944,Y 131.6856,Z 161,A 92.878,B 16.7028,C -0.4423,E1 16.6966,E2 716.0958} C_DIS
LIN {X -13.3832,Y 131.3128,Z 161,A 94.8055,B 16.7028,C -0.4421,E1 16.6912,E2 714.1676} C_DIS
LIN {X -17.7941,Y 130.7875,Z 161,A 96.7135,B 16.7028,C -0.4404,E1 16.6859,E2 712.2633} C_DIS
LIN {X -21.1135,Y 130.2926,Z 161,A 98.7458,B 16.7023,C -0.459,E1 16.6802,E2 710.1636} C_DIS
LIN {X -26.198,Y 129.3648,Z 161,A 100.0234,B 16.7031,C -0.425,E1 16.677,E2 709.0021} C_DIS
LIN {X -31.8217,Y 128.0976,Z 161,A 103.001,B 16.7028,C -0.4388,E1 16.6687,E2 705.9705} C_DIS
LIN {X -36.0351,Y 126.9774,Z 161,A 105.5004,B 16.7023,C -0.4573,E1 16.6618,E2 703.4005} C_DIS
LIN {X -41.4918,Y 125.2996,Z 161,A 107.3001,B 16.703,C -0.4321,E1 16.6572,E2 701.6837} C_DIS
LIN {X -45.846,Y 123.7735,Z 161,A 109.1619,B 16.7031,C -0.4251,E1 16.6524,E2 699.8404} C_DIS
LIN {X -49.1516,Y 122.4976,Z 161,A 110.7171,B 16.7031,C -0.4238,E1 16.6484,E2 698.2846} C_DIS
LIN {X -56.5208,Y 119.2772,Z 161,A 114.0915,B 16.7034,C -0.4153,E1 16.6398,E2 694.9276} C_DIS
LIN {X -64.0853,Y 115.3911,Z 161,A 118.006,B 16.7034,C -0.4168,E1 16.6301,E2 690.9911} C_DIS
LIN {X -67.5958,Y 113.3703,Z 161,A 119.7914,B 16.7034,C -0.4148,E1 16.6257,E2 689.2045} C_DIS
LIN {X -70.1623,Y 111.8006,Z 161,A 121.1793,B 16.7034,C -0.4152,E1 16.6224,E2 687.8084} C_DIS
LIN {X -74.0635,Y 109.2548,Z 161,A 123.2133,B 16.7034,C -0.4119,E1 16.6177,E2 685.7753} C_DIS
LIN {X -78.9066,Y 105.81,Z 161,A 125.7561,B 16.7036,C -0.4059,E1 16.612,E2 683.2399} C_DIS
LIN {X -82.4839,Y 103.0463,Z 161,A 128.4408,B 16.7031,C -0.4253,E1 16.6059,E2 680.4718} C_DIS
LIN {X -86.8645,Y 99.3809,Z 161,A 130.2254,B 16.7038,C -0.3977,E1 16.6023,E2 678.7729} C_DIS
LIN {X -90.0569,Y 96.4975,Z 161,A 132.1038,B 16.7038,C -0.394,E1 16.5985,E2 676.8956} C_DIS
LIN {X -92.4772,Y 94.1806,Z 161,A 133.7938,B 16.7038,C -0.3983,E1 16.595,E2 675.1795} C_DIS
LIN {X -94.7588,Y 91.8846,Z 161,A 135.1643,B 16.7038,C -0.394,E1 16.5924,E2 673.8149} C_DIS
LIN {X -98.3669,Y 88.0112,Z 161,A 137.3267,B 16.7041,C -0.3843,E1 16.5884,E2 671.6716} C_DIS
LIN {X -101.3182,Y 84.5974,Z 161,A 139.3904,B 16.7041,C -0.3829,E1 16.5846,E2 669.5982} C_DIS
LIN {X -104.4621,Y 80.6828,Z 161,A 141.5888,B 16.7042,C -0.3781,E1 16.5808,E2 667.4005} C_DIS
LIN {X -107.4861,Y 76.608,Z 161,A 143.6314,B 16.7045,C -0.3675,E1 16.5775,E2 665.3798} C_DIS
LIN {X -109.0791,Y 74.323,Z 161,A 145.1803,B 16.7043,C -0.375,E1 16.575,E2 663.7925} C_DIS
LIN {X -110.9891,Y 71.4389,Z 161,A 146.3372,B 16.7046,C -0.3602,E1 16.5733,E2 662.6784} C_DIS
LIN {X -113.5584,Y 67.2802,Z 161,A 148.5921,B 16.7046,C -0.3587,E1 16.57,E2 660.4108} C_DIS
LIN {X -115.7308,Y 63.4703,Z 161,A 150.3108,B 16.7049,C -0.3477,E1 16.5677,E2 658.7165} C_DIS
LIN {X -117.6338,Y 59.8645,Z 161,A 152.2783,B 16.7049,C -0.349,E1 16.5651,E2 656.7281} C_DIS
LIN {X -119.598,Y 55.8393,Z 161,A 154.1458,B 16.705,C -0.3411,E1 16.5629,E2 654.8726} C_DIS
LIN {X -120.8363,Y 53.1103,Z 161,A 155.6175,B 16.705,C -0.3428,E1 16.5612,E2 653.3825} C_DIS
LIN {X -122.2336,Y 49.8065,Z 161,A 156.899,B 16.7052,C -0.3297,E1 16.5599,E2 652.1357} C_DIS
LIN {X -123.4565,Y 46.6925,Z 161,A 158.4003,B 16.7052,C -0.327,E1 16.5584,E2 650.6308} C_DIS
LIN {X -124.6414,Y 43.4291,Z 161,A 160.0314,B 16.7053,C -0.3265,E1 16.5568,E2 648.9872} C_DIS
LIN {X -125.9444,Y 39.4954,Z 161,A 161.9887,B 16.7053,C -0.3261,E1 16.5551,E2 647.0138} C_DIS
LIN {X -127.0525,Y 35.7664,Z 161,A 163.5734,B 16.7055,C -0.3178,E1 16.5539,E2 645.4437} C_DIS
LIN {X -128.0158,Y 32.15,Z 161,A 165.2665,B 16.7055,C -0.3151,E1 16.5527,E2 643.7448} C_DIS
LIN {X -128.703,Y 29.2761,Z 161,A 166.7538,B 16.7055,C -0.3176,E1 16.5518,E2 642.2351} C_DIS
LIN {X -129.7591,Y 24.177,Z 161,A 169.3178,B 16.7055,C -0.3203,E1 16.5504,E2 639.6382} C_DIS
LIN {X -130.5089,Y 19.7285,Z 161,A 170.8597,B 16.7058,C -0.3013,E1 16.5498,E2 638.1486} C_DIS
LIN {X -131.0263,Y 15.9304,Z 161,A 172.478,B 16.7058,C -0.2948,E1 16.5492,E2 636.538} C_DIS
LIN {X -131.3866,Y 12.616,Z 161,A 174.3674,B 16.7058,C -0.3042,E1 16.5487,E2 634.598} C_DIS
LIN {X -131.723,Y 8.4109,Z 161,A 175.7886,B 16.706,C -0.2858,E1 16.5485,E2 633.2282} C_DIS
LIN {X -131.9021,Y 4.853,Z 161,A 177.8607,B 16.7058,C -0.2975,E1 16.5482,E2 631.0955} C_DIS
LIN {X -131.9926,Y 0.1569,Z 161,A 179.9073,B 16.7059,C -0.2914,E1 16.5482,E2 629.0508} C_DIS
LIN {X -131.9191,Y -4.4135,Z 161,A -178.4969,B 16.7062,C -0.2732,E1 16.5484,E2 627.5041} C_DIS
LIN {X -131.7154,Y -8.5344,Z 161,A -176.1359,B 16.706,C -0.2857,E1 16.5488,E2 625.0773} C_DIS
LIN {X -131.2681,Y -13.7985,Z 161,A -174.2803,B 16.7064,C -0.2649,E1 16.5493,E2 623.277} C_DIS
LIN {X -130.4421,Y -20.1601,Z 161,A -171.677,B 16.7066,C -0.2509,E1 16.5503,E2 620.6989} C_DIS
LIN {X -129.99,Y -22.8976,Z 161,A -170.1389,B 16.7065,C -0.2577,E1 16.5511,E2 619.1225} C_DIS
LIN {X -129.3374,Y -26.3327,Z 161,A -168.5389,B 16.7065,C -0.2558,E1 16.5519,E2 617.5145} C_DIS
LIN {X -128.4808,Y -30.2446,Z 161,A -167.2201,B 16.7068,C -0.2375,E1 16.5527,E2 616.248} C_DIS
LIN {X -127.607,Y -33.7353,Z 161,A -165.6364,B 16.7068,C -0.2336,E1 16.5538,E2 614.6635} C_DIS
LIN {X -126.835,Y -36.5343,Z 161,A -164.4529,B 16.7068,C -0.2275,E1 16.5547,E2 613.4906} C_DIS
LIN {X -125.8458,Y -39.8058,Z 161,A -162.8339,B 16.7068,C -0.2275,E1 16.5561,E2 611.8572} C_DIS
LIN {X -124.7831,Y -43.0202,Z 161,A -161.385,B 16.707,C -0.2227,E1 16.5574,E2 610.4124} C_DIS
LIN {X -123.79,Y -45.8019,Z 161,A -160.1114,B 16.707,C -0.2188,E1 16.5586,E2 609.1412} C_DIS
LIN {X -122.39,Y -49.4184,Z 161,A -158.2954,B 16.707,C -0.2183,E1 16.5605,E2 607.3111} C_DIS
LIN {X -121.2221,Y -52.2181,Z 161,A -156.7108,B 16.707,C -0.2231,E1 16.5623,E2 605.6959} C_DIS
LIN {X -119.7973,Y -55.4085,Z 161,A -155.0312,B 16.707,C -0.2242,E1 16.5643,E2 603.9982} C_DIS
LIN {X -117.9043,Y -59.3331,Z 161,A -153.5507,B 16.7072,C -0.2061,E1 16.566,E2 602.569} C_DIS
LIN {X -116.1202,Y -62.7551,Z 161,A -151.8402,B 16.7072,C -0.2028,E1 16.5683,E2 600.856} C_DIS
LIN {X -113.7015,Y -67.0374,Z 161,A -149.6922,B 16.7072,C -0.1977,E1 16.5713,E2 598.7083} C_DIS
LIN {X -112.1236,Y -69.6442,Z 161,A -148.3131,B 16.7072,C -0.1961,E1 16.5733,E2 597.3237} C_DIS
LIN {X -109.7074,Y -73.3915,Z 161,A -146.5551,B 16.7074,C -0.1857,E1 16.576,E2 595.5886} C_DIS
LIN {X -107.733,Y -76.2605,Z 161,A -144.8844,B 16.7074,C -0.1871,E1 16.5787,E2 593.9002} C_DIS
LIN {X -105.0813,Y -79.8754,Z 161,A -142.9699,B 16.7074,C -0.1815,E1 16.5818,E2 591.991} C_DIS
LIN {X -102.3821,Y -83.3066,Z 161,A -141.0512,B 16.7074,C -0.1779,E1 16.5852,E2 590.0708} C_DIS
LIN {X -99.9129,Y -86.2522,Z 161,A -139.0246,B 16.7074,C -0.1858,E1 16.589,E2 588.0022} C_DIS
LIN {X -97.3936,Y -89.0875,Z 161,A -137.6429,B 16.7075,C -0.1737,E1 16.5915,E2 586.6536} C_DIS
LIN {X -94.2519,Y -92.4044,Z 161,A -135.7221,B 16.7075,C -0.1675,E1 16.5952,E2 584.7416} C_DIS
LIN {X -91.3215,Y -95.3017,Z 161,A -133.9599,B 16.7076,C -0.163,E1 16.5987,E2 582.9836} C_DIS
LIN {X -88.2281,Y -98.1726,Z 161,A -132.2008,B 16.7076,C -0.157,E1 16.6023,E2 581.2343} C_DIS
LIN {X -84.2949,Y -101.5691,Z 161,A -129.5357,B 16.7076,C -0.1663,E1 16.6081,E2 578.521} C_DIS
LIN {X -81.6451,Y -103.7116,Z 161,A -128.3479,B 16.7077,C -0.1541,E1 16.6106,E2 577.369} C_DIS
LIN {X -79.163,Y -105.6191,Z 161,A -126.768,B 16.7077,C -0.159,E1 16.6142,E2 575.763} C_DIS
LIN {X -76.4141,Y -107.6246,Z 161,A -125.2714,B 16.7077,C -0.1572,E1 16.6176,E2 574.2647} C_DIS
LIN {X -72.3361,Y -110.4064,Z 161,A -123.2555,B 16.7077,C -0.1496,E1 16.6223,E2 572.2649} C_DIS
LIN {X -68.53,Y -112.8083,Z 161,A -121.2981,B 16.7077,C -0.1469,E1 16.6269,E2 570.3077} C_DIS
LIN {X -64.6522,Y -115.0743,Z 161,A -119.4521,B 16.7078,C -0.1407,E1 16.6313,E2 568.4746} C_DIS
LIN {X -61.5139,Y -116.7799,Z 161,A -117.9072,B 16.7078,C -0.1386,E1 16.6351,E2 566.9306} C_DIS
LIN {X -58.7607,Y -118.1898,Z 161,A -116.4971,B 16.7078,C -0.1392,E1 16.6387,E2 565.5127} C_DIS
LIN {X -55.5236,Y -119.744,Z 161,A -114.9876,B 16.7078,C -0.1357,E1 16.6425,E2 564.0093} C_DIS
LIN {X -52.5082,Y -121.0967,Z 161,A -113.6779,B 16.7079,C -0.13,E1 16.6458,E2 562.7148} C_DIS
LIN {X -49.6483,Y -122.2974,Z 161,A -112.1977,B 16.7079,C -0.1331,E1 16.6496,E2 561.2185} C_DIS
LIN {X -46.2983,Y -123.6041,Z 161,A -110.6719,B 16.7079,C -0.1304,E1 16.6536,E2 559.6971} C_DIS
LIN {X -43.3739,Y -124.6605,Z 161,A -109.2607,B 16.7079,C -0.1313,E1 16.6573,E2 558.2784} C_DIS
LIN {X -36.076,Y -126.966,Z 161,A -104.9068,B 16.7076,C -0.1644,E1 16.6693,E2 553.7981} C_DIS
LIN {X -29.2992,Y -128.6978,Z 161,A -102.8639,B 16.7079,C -0.1284,E1 16.6746,E2 551.8764} C_DIS
LIN {X -25.108,Y -129.5811,Z 161,A -100.9498,B 16.7079,C -0.1294,E1 16.6798,E2 549.9553} C_DIS
LIN {X -21.2935,Y -130.2626,Z 161,A -99.2291,B 16.7079,C -0.1302,E1 16.6846,E2 548.2295} C_DIS
LIN {X -17.2213,Y -130.8626,Z 161,A -97.5463,B 16.7079,C -0.1261,E1 16.6892,E2 546.5588} C_DIS
LIN {X -13.2365,Y -131.327,Z 161,A -95.731,B 16.7079,C -0.1284,E1 16.6943,E2 544.734} C_DIS
LIN {X -9.571,Y -131.6435,Z 161,A -94.1359,B 16.7079,C -0.1282,E1 16.6987,E2 543.1384} C_DIS
LIN {X -5.1589,Y -131.8901,Z 161,A -92.2703,B 16.7079,C -0.1264,E1 16.7039,E2 541.2784} C_DIS
LIN {X -0.9248,Y -131.988,Z 161,A -90.4592,B 16.7079,C -0.1257,E1 16.7089,E2 539.4699} C_DIS
LIN {X -0.9248,Y -131.988,Z 161,A -90.4592,B 16.7079,C -0.1257,E1 16.7089,E2 539.4699} C_DIS
Enddeposition()
LIN {X 0.9263,Y -131.0637,Z 161,A -89.5349,B 14.0867,C 0.1068,E1 14.0879,E2 539.3172} C_DIS
Startdeposition()
$VEL.CP = VEL_PRINT
LIN {X -3.109,Y -131.031,Z 161,A -91.3335,B 14.0867,C 0.108,E1 14.0829,E2 541.1208} C_DIS
LIN {X -7.1773,Y -130.8715,Z 161,A -93.0229,B 14.0867,C 0.1055,E1 14.0782,E2 542.8002} C_DIS
LIN {X -10.4222,Y -130.6531,Z 161,A -94.5813,B 14.0867,C 0.1093,E1 14.0738,E2 544.3754} C_DIS
LIN {X -14.445,Y -130.269,Z 161,A -96.2497,B 14.0867,C 0.1062,E1 14.0692,E2 546.0327} C_DIS
LIN {X -17.4037,Y -129.9066,Z 161,A -97.6483,B 14.0867,C 0.1086,E1 14.0653,E2 547.4431} C_DIS
LIN {X -21.718,Y -129.2548,Z 161,A -99.4781,B 14.0867,C 0.1058,E1 14.0603,E2 549.2642} C_DIS
LIN {X -25.7301,Y -128.5168,Z 161,A -101.7622,B 14.0867,C 0.1192,E1 14.0539,E2 551.608} C_DIS
LIN {X -29.9772,Y -127.5946,Z 161,A -103.1284,B 14.0867,C 0.1032,E1 14.0503,E2 552.9116} C_DIS
LIN {X -34.6708,Y -126.3993,Z 161,A -105.38,B 14.0867,C 0.1056,E1 14.0442,E2 555.1794} C_DIS
LIN {X -39.5959,Y -124.9426,Z 161,A -107.3233,B 14.0868,C 0.0955,E1 14.0391,E2 557.0872} C_DIS
LIN {X -44.3307,Y -123.3418,Z 161,A -109.7286,B 14.0868,C 0.0999,E1 14.0327,E2 559.5188} C_DIS
LIN {X -48.0159,Y -121.9556,Z 161,A -111.4378,B 14.0868,C 0.0979,E1 14.0282,E2 561.2267} C_DIS
LIN {X -50.6567,Y -120.8814,Z 161,A -112.6997,B 14.0868,C 0.0971,E1 14.025,E2 562.4903} C_DIS
LIN {X -53.7452,Y -119.5403,Z 161,A -114.1725,B 14.0868,C 0.0955,E1 14.0212,E2 563.9632} C_DIS
LIN {X -56.8425,Y -118.0993,Z 161,A -115.6674,B 14.0868,C 0.0939,E1 14.0174,E2 565.4582} C_DIS
LIN {X -60.1736,Y -116.4394,Z 161,A -117.4677,B 14.0868,C 0.0966,E1 14.0129,E2 567.2789} C_DIS
LIN {X -64.1303,Y -114.3075,Z 161,A -119.3834,B 14.0868,C 0.0927,E1 14.0082,E2 569.1885} C_DIS
LIN {X -67.9172,Y -112.0988,Z 161,A -121.1483,B 14.0868,C 0.0859,E1 14.004,E2 570.9351} C_DIS
LIN {X -70.6543,Y -110.3941,Z 161,A -122.7173,B 14.0868,C 0.0881,E1 14.0003,E2 572.5226} C_DIS
LIN {X -74.394,Y -107.9096,Z 161,A -124.6274,B 14.0868,C 0.0837,E1 13.9959,E2 574.426} C_DIS
LIN {X -77.4018,Y -105.7729,Z 161,A -126.3497,B 14.0868,C 0.084,E1 13.9919,E2 576.1606} C_DIS
LIN {X -80.5832,Y -103.37,Z 161,A -129.1329,B 14.0868,C 0.1086,E1 13.9856,E2 579.0645} C_DIS
LIN {X -86.3589,Y -98.5955,Z 161,A -131.3251,B 14.0869,C 0.0739,E1 13.9812,E2 581.1292} C_DIS
LIN {X -90.4624,Y -94.8444,Z 161,A -133.6473,B 14.0869,C 0.0663,E1 13.9764,E2 583.4376} C_DIS
LIN {X -92.8662,Y -92.492,Z 161,A -135.3106,B 14.0869,C 0.0685,E1 13.9731,E2 585.1229} C_DIS
LIN {X -95.9506,Y -89.2881,Z 161,A -137.6307,B 14.0869,C 0.0743,E1 13.9686,E2 587.486} C_DIS
LIN {X -98.6411,Y -86.3067,Z 161,A -138.8418,B 14.087,C 0.0563,E1 13.9665,E2 588.6323} C_DIS
LIN {X -101.099,Y -83.4142,Z 161,A -140.8023,B 14.087,C 0.0605,E1 13.9629,E2 590.6271} C_DIS
LIN {X -103.6934,Y -80.166,Z 161,A -142.569,B 14.087,C 0.0551,E1 13.9598,E2 592.3868} C_DIS
LIN {X -105.9403,Y -77.1728,Z 161,A -144.1082,B 14.087,C 0.0487,E1 13.9573,E2 593.9135} C_DIS
LIN {X -108.2844,Y -73.8479,Z 161,A -145.8088,B 14.087,C 0.0425,E1 13.9546,E2 595.6039} C_DIS
LIN {X -110.1952,Y -70.965,Z 161,A -147.5465,B 14.087,C 0.0446,E1 13.9519,E2 597.3669} C_DIS
LIN {X -112.0393,Y -68.0157,Z 161,A -149.0688,B 14.087,C 0.0409,E1 13.9497,E2 598.8882} C_DIS
LIN {X -114.3144,Y -64.1181,Z 161,A -151.0663,B 14.087,C 0.0365,E1 13.9469,E2 600.887} C_DIS
LIN {X -116.2673,Y -60.5022,Z 161,A -152.7602,B 14.087,C 0.0292,E1 13.9447,E2 602.5674} C_DIS
LIN {X -119.6048,Y -53.6011,Z 161,A -155.846,B 14.0871,C 0.0136,E1 13.9411,E2 605.6193} C_DIS
LIN {X -121.241,Y -49.7956,Z 161,A -158.2762,B 14.0871,C 0.0246,E1 13.9383,E2 608.1202} C_DIS
LIN {X -122.4229,Y -46.8139,Z 161,A -159.5369,B 14.0871,C 0.0171,E1 13.9371,E2 609.3632} C_DIS
LIN {X -123.862,Y -42.8556,Z 161,A -161.2902,B 14.0871,C 0.0097,E1 13.9354,E2 611.1044} C_DIS
LIN {X -125.0653,Y -39.2118,Z 161,A -163.103,B 14.0871,C 0.0085,E1 13.9339,E2 612.9314} C_DIS
LIN {X -126.2975,Y -35.0348,Z 161,A -164.864,B 14.0871,C -0.0006,E1 13.9325,E2 614.6738} C_DIS
LIN {X -127.1709,Y -31.722,Z 161,A -166.486,B 14.0871,C -0.0017,E1 13.9314,E2 616.3088} C_DIS
LIN {X -128.1576,Y -27.4609,Z 161,A -168.325,B 14.0871,C -0.0091,E1 13.9303,E2 618.1373} C_DIS
LIN {X -128.7135,Y -24.7242,Z 161,A -169.5935,B 14.0871,C -0.0115,E1 13.9296,E2 619.41} C_DIS
LIN {X -129.4199,Y -20.7219,Z 161,A -171.4412,B 14.0871,C -0.0149,E1 13.9288,E2 621.2641} C_DIS
LIN {X -130.1982,Y -15.0706,Z 161,A -173.8146,B 14.0871,C -0.0253,E1 13.9279,E2 623.6207} C_DIS
LIN {X -130.6524,Y -10.4313,Z 161,A -176.1892,B 14.0871,C -0.0229,E1 13.9273,E2 626.032} C_DIS
LIN {X -130.9118,Y -6.3761,Z 161,A -178.0719,B 14.0871,C -0.0255,E1 13.927,E2 627.9249} C_DIS
LIN {X -131.0344,Y -2.9222,Z 161,A -179.4136,B 14.0871,C -0.0343,E1 13.927,E2 629.2453} C_DIS
LIN {X -131.0422,Y 2.5724,Z 161,A 178.0231,B 14.0871,C -0.0374,E1 13.927,E2 631.8243} C_DIS
LIN {X -130.9372,Y 5.8692,Z 161,A 176.2595,B 14.0871,C -0.0337,E1 13.9272,E2 633.6233} C_DIS
LIN {X -130.6433,Y 10.5385,Z 161,A 174.7785,B 14.0871,C -0.0539,E1 13.9275,E2 635.0368} C_DIS
LIN {X -130.3169,Y 13.9992,Z 161,A 173.2314,B 14.0871,C -0.0578,E1 13.928,E2 636.5852} C_DIS
LIN {X -129.8393,Y 17.9061,Z 161,A 171.5996,B 14.087,C -0.0651,E1 13.9285,E2 638.2046} C_DIS
LIN {X -129.4051,Y 20.8176,Z 161,A 170.0364,B 14.087,C -0.062,E1 13.9292,E2 639.7982} C_DIS
LIN {X -128.5623,Y 25.5069,Z 161,A 168.1932,B 14.087,C -0.0742,E1 13.9302,E2 641.6111} C_DIS
LIN {X -127.9249,Y 28.5325,Z 161,A 166.6137,B 14.087,C -0.0725,E1 13.9311,E2 643.2152} C_DIS
LIN {X -127.0398,Y 32.2385,Z 161,A 165.0596,B 14.0869,C -0.0802,E1 13.9321,E2 644.7542} C_DIS
LIN {X -126.1523,Y 35.5539,Z 161,A 163.6042,B 14.0869,C -0.0857,E1 13.9332,E2 646.2026} C_DIS
LIN {X -125.0954,Y 39.1173,Z 161,A 161.9245,B 14.0869,C -0.089,E1 13.9346,E2 647.8867} C_DIS
LIN {X -124.0697,Y 42.2565,Z 161,A 160.495,B 14.0869,C -0.0935,E1 13.9358,E2 649.3127} C_DIS
LIN {X -122.8867,Y 45.5788,Z 161,A 158.7903,B 14.0869,C -0.0938,E1 13.9375,E2 651.0341} C_DIS
LIN {X -121.5491,Y 49.0327,Z 161,A 157.1746,B 14.0868,C -0.0985,E1 13.9391,E2 652.6473} C_DIS
LIN {X -120.2254,Y 52.1944,Z 161,A 155.6942,B 14.0868,C -0.1031,E1 13.9407,E2 654.1238} C_DIS
LIN {X -118.8059,Y 55.3505,Z 161,A 154.099,B 14.0868,C -0.1052,E1 13.9426,E2 655.7265} C_DIS
LIN {X -117.3035,Y 58.4683,Z 161,A 152.619,B 14.0867,C -0.1101,E1 13.9444,E2 657.2009} C_DIS
LIN {X -115.1453,Y 62.6137,Z 161,A 150.6644,B 14.0867,C -0.1179,E1 13.947,E2 659.1427} C_DIS
LIN {X -113.3541,Y 65.801,Z 161,A 148.8759,B 14.0867,C -0.1173,E1 13.9495,E2 660.9511} C_DIS
LIN {X -111.6737,Y 68.614,Z 161,A 147.4944,B 14.0866,C -0.1223,E1 13.9515,E2 662.3249} C_DIS
LIN {X -109.5023,Y 72.0287,Z 161,A 145.7011,B 14.0866,C -0.1262,E1 13.9542,E2 664.1189} C_DIS
LIN {X -107.2595,Y 75.3284,Z 161,A 144.0112,B 14.0866,C -0.132,E1 13.9568,E2 665.8004} C_DIS
LIN {X -103.8797,Y 79.9239,Z 161,A 141.3917,B 14.0865,C -0.1349,E1 13.9612,E2 668.4313} C_DIS
LIN {X -101.0851,Y 83.431,Z 161,A 139.4596,B 14.0865,C -0.1403,E1 13.9646,E2 670.3577} C_DIS
LIN {X -98.4027,Y 86.5788,Z 161,A 137.5998,B 14.0865,C -0.1432,E1 13.968,E2 672.2214} C_DIS
LIN {X -95.7079,Y 89.5487,Z 161,A 135.8246,B 14.0864,C -0.1466,E1 13.9714,E2 673.9969} C_DIS
LIN {X -93.0776,Y 92.2793,Z 161,A 134.2984,B 14.0863,C -0.1536,E1 13.9743,E2 675.5061} C_DIS
LIN {X -90.4904,Y 94.8176,Z 161,A 132.6348,B 14.0863,C -0.155,E1 13.9777,E2 677.1771} C_DIS
LIN {X -87.7846,Y 97.3288,Z 161,A 130.9936,B 14.0863,C -0.1576,E1 13.9811,E2 678.8195} C_DIS
LIN {X -85.0466,Y 99.7296,Z 161,A 129.1873,B 14.0863,C -0.1553,E1 13.9849,E2 680.6486} C_DIS
LIN {X -81.3094,Y 102.8,Z 161,A 127.237,B 14.0862,C -0.1637,E1 13.9891,E2 682.5778} C_DIS
LIN {X -78.2587,Y 105.1402,Z 161,A 125.1612,B 14.0862,C -0.1565,E1 13.9939,E2 684.6969} C_DIS
LIN {X -75.0659,Y 107.4433,Z 161,A 123.8914,B 14.0861,C -0.1714,E1 13.9966,E2 685.9133} C_DIS
LIN {X -72.2653,Y 109.3465,Z 161,A 122.1209,B 14.0861,C -0.1664,E1 14.0008,E2 687.7155} C_DIS
LIN {X -67.8737,Y 112.1251,Z 161,A 120.0015,B 14.0861,C -0.1741,E1 14.0058,E2 689.8151} C_DIS
LIN {X -64.1147,Y 114.3163,Z 161,A 117.615,B 14.0861,C -0.1643,E1 14.0117,E2 692.255} C_DIS
LIN {X -60.1064,Y 116.4736,Z 161,A 116.226,B 14.086,C -0.1831,E1 14.015,E2 693.5734} C_DIS
LIN {X -57.5447,Y 117.7591,Z 161,A 114.9297,B 14.086,C -0.1838,E1 14.0182,E2 694.8735} C_DIS
LIN {X -53.9359,Y 119.455,Z 161,A 112.8666,B 14.086,C -0.1775,E1 14.0236,E2 696.9717} C_DIS
LIN {X -50.9722,Y 120.7496,Z 161,A 111.8833,B 14.0859,C -0.1908,E1 14.026,E2 697.9044} C_DIS
LIN {X -48.5858,Y 121.7292,Z 161,A 110.6186,B 14.0859,C -0.1885,E1 14.0293,E2 699.1839} C_DIS
LIN {X -45.5948,Y 122.8807,Z 161,A 109.1941,B 14.0859,C -0.1895,E1 14.033,E2 700.6098} C_DIS
LIN {X -39.6204,Y 124.9348,Z 161,A 106.4607,B 14.0859,C -0.1931,E1 14.0402,E2 703.3377} C_DIS
LIN {X -36.4273,Y 125.9033,Z 161,A 104.975,B 14.0859,C -0.1937,E1 14.0442,E2 704.8254} C_DIS
LIN {X -32.741,Y 126.9122,Z 161,A 102.5834,B 14.086,C -0.1756,E1 14.0509,E2 707.2981} C_DIS
LIN {X -27.6185,Y 128.1236,Z 161,A 101.1102,B 14.0857,C -0.1998,E1 14.0546,E2 708.675} C_DIS
LIN {X -20.5586,Y 129.4452,Z 161,A 97.9251,B 14.0857,C -0.2005,E1 14.0634,E2 711.8634} C_DIS
LIN {X -17.1455,Y 129.9404,Z 161,A 96.2519,B 14.0857,C -0.1966,E1 14.0681,E2 713.5546} C_DIS
LIN {X -12.5888,Y 130.4608,Z 161,A 94.2064,B 14.0857,C -0.1963,E1 14.0738,E2 715.6036} C_DIS
LIN {X -8.07,Y 130.8181,Z 161,A 92.3092,B 14.0857,C -0.1993,E1 14.079,E2 717.49} C_DIS
LIN {X -4.2182,Y 131.0002,Z 161,A 90.6132,B 14.0857,C -0.1993,E1 14.0838,E2 719.1864} C_DIS
LIN {X -0.0002,Y 131.0689,Z 161,A 88.7959,B 14.0857,C -0.2002,E1 14.0888,E2 720.9997} C_DIS
LIN {X 3.0129,Y 131.0337,Z 161,A 87.3647,B 14.0857,C -0.1971,E1 14.0928,E2 722.4435} C_DIS
LIN {X 6.8033,Y 130.8903,Z 161,A 85.844,B 14.0857,C -0.2009,E1 14.097,E2 723.9476} C_DIS
LIN {X 10.2889,Y 130.6644,Z 161,A 84.344,B 14.0857,C -0.2014,E1 14.1012,E2 725.444} C_DIS
LIN {X 13.941,Y 130.3232,Z 161,A 82.644,B 14.0857,C -0.1984,E1 14.106,E2 727.1544} C_DIS
LIN {X 18.3196,Y 129.7802,Z 161,A 80.7072,B 14.0857,C -0.1976,E1 14.1113,E2 729.0916} C_DIS
LIN {X 22.4647,Y 129.1286,Z 161,A 78.3977,B 14.086,C -0.1832,E1 14.1178,E2 731.4552} C_DIS
LIN {X 26.908,Y 128.277,Z 161,A 77,B 14.0857,C -0.1988,E1 14.1215,E2 732.7858} C_DIS
LIN {X 29.8109,Y 127.6329,Z 161,A 75.6869,B 14.0857,C -0.1977,E1 14.1251,E2 734.1001} C_DIS
LIN {X 33.6458,Y 126.6744,Z 161,A 73.649,B 14.0859,C -0.1876,E1 14.1307,E2 736.1735} C_DIS
LIN {X 36.7493,Y 125.809,Z 161,A 72.4611,B 14.0859,C -0.1929,E1 14.1338,E2 737.3358} C_DIS
LIN {X 40.9076,Y 124.5201,Z 161,A 70.577,B 14.0859,C -0.1919,E1 14.1388,E2 739.2176} C_DIS
LIN {X 45.0523,Y 123.0816,Z 161,A 68.7449,B 14.0859,C -0.1926,E1 14.1436,E2 741.0396} C_DIS
LIN {X 47.6692,Y 122.0904,Z 161,A 67.5222,B 14.0859,C -0.1914,E1 14.1468,E2 742.2622} C_DIS
LIN {X 50.6704,Y 120.8756,Z 161,A 66.1002,B 14.0859,C -0.1897,E1 14.1504,E2 743.685} C_DIS
LIN {X 53.9844,Y 119.4334,Z 161,A 64.5518,B 14.0859,C -0.1889,E1 14.1544,E2 745.2298} C_DIS
LIN {X 57.4395,Y 117.811,Z 161,A 62.9654,B 14.0859,C -0.1893,E1 14.1584,E2 746.8069} C_DIS
LIN {X 59.6228,Y 116.7198,Z 161,A 61.7753,B 14.0859,C -0.1843,E1 14.1614,E2 748.0113} C_DIS
LIN {X 62.9902,Y 114.9399,Z 161,A 60.255,B 14.0859,C -0.1863,E1 14.1651,E2 749.5151} C_DIS
LIN {X 65.0824,Y 113.7681,Z 161,A 59.2084,B 14.0859,C -0.1849,E1 14.1676,E2 750.5617} C_DIS
LIN {X 67.6439,Y 112.2641,Z 161,A 57.9191,B 14.0859,C -0.1833,E1 14.1707,E2 751.8502} C_DIS
LIN {X 70.3048,Y 110.6177,Z 161,A 56.1757,B 14.0861,C -0.17,E1 14.1749,E2 753.6375} C_DIS
LIN {X 74.0489,Y 108.1465,Z 161,A 54.389,B 14.0861,C -0.1721,E1 14.179,E2 755.4045} C_DIS
LIN {X 76.7936,Y 106.2151,Z 161,A 53.0552,B 14.0861,C -0.1736,E1 14.182,E2 756.7233} C_DIS
LIN {X 79.9294,Y 103.8765,Z 161,A 51.2298,B 14.0861,C -0.1672,E1 14.1861,E2 758.5626} C_DIS
LIN {X 83.3673,Y 101.1378,Z 161,A 49.3319,B 14.0861,C -0.1644,E1 14.1902,E2 760.4585} C_DIS
LIN {X 86.7243,Y 98.2741,Z 161,A 47.4768,B 14.0861,C -0.163,E1 14.1941,E2 762.3058} C_DIS
LIN {X 89.6486,Y 95.6147,Z 161,A 45.7555,B 14.0862,C -0.1598,E1 14.1977,E2 764.0271} C_DIS
LIN {X 92.4533,Y 92.9047,Z 161,A 44.0288,B 14.0862,C -0.1557,E1 14.2011,E2 765.7572} C_DIS
LIN {X 95.6043,Y 89.6596,Z 161,A 42.0309,B 14.0863,C -0.1509,E1 14.205,E2 767.7586} C_DIS
LIN {X 98.5099,Y 86.457,Z 161,A 40.1485,B 14.0863,C -0.147,E1 14.2085,E2 769.6412} C_DIS
LIN {X 101.4085,Y 83.0374,Z 161,A 38.3097,B 14.0863,C -0.1463,E1 14.2117,E2 771.467} C_DIS
LIN {X 103.887,Y 79.9156,Z 161,A 36.5413,B 14.0864,C -0.1415,E1 14.2148,E2 773.2395} C_DIS
LIN {X 106.745,Y 76.0554,Z 161,A 34.528,B 14.0864,C -0.1392,E1 14.2181,E2 775.2442} C_DIS
LIN {X 108.9027,Y 72.9323,Z 161,A 32.9846,B 14.0864,C -0.1388,E1 14.2205,E2 776.7751} C_DIS
LIN {X 110.608,Y 70.3202,Z 161,A 31.3875,B 14.0865,C -0.1282,E1 14.223,E2 778.4007} C_DIS
LIN {X 112.9524,Y 66.488,Z 161,A 29.6832,B 14.0865,C -0.1313,E1 14.2254,E2 780.076} C_DIS
LIN {X 114.2029,Y 64.3164,Z 161,A 28.5976,B 14.0865,C -0.1289,E1 14.2269,E2 781.1613} C_DIS
LIN {X 115.3796,Y 62.181,Z 161,A 27.2469,B 14.0866,C -0.1172,E1 14.2287,E2 782.5463} C_DIS
LIN {X 117.1438,Y 58.79,Z 161,A 25.6367,B 14.0866,C -0.1147,E1 14.2307,E2 784.1508} C_DIS
LIN {X 119.0497,Y 54.8233,Z 161,A 23.8975,B 14.0866,C -0.1154,E1 14.2328,E2 785.8699} C_DIS
LIN {X 120.3971,Y 51.7975,Z 161,A 22.4727,B 14.0866,C -0.1122,E1 14.2344,E2 787.2933} C_DIS
LIN {X 121.7141,Y 48.6233,Z 161,A 20.971,B 14.0867,C -0.1081,E1 14.236,E2 788.7963} C_DIS
LIN {X 122.8344,Y 45.7184,Z 161,A 19.6686,B 14.0867,C -0.1062,E1 14.2373,E2 790.0931} C_DIS
LIN {X 123.8489,Y 42.8935,Z 161,A 17.8495,B 14.0869,C -0.0866,E1 14.239,E2 791.9729} C_DIS
LIN {X 125.1579,Y 38.9133,Z 161,A 16.5242,B 14.0868,C -0.0973,E1 14.2401,E2 793.2407} C_DIS
LIN {X 126.1353,Y 35.6148,Z 161,A 14.9507,B 14.0868,C -0.0908,E1 14.2413,E2 794.8239} C_DIS
LIN {X 127.0697,Y 32.1205,Z 161,A 13.4532,B 14.0868,C -0.0889,E1 14.2423,E2 796.3132} C_DIS
LIN {X 127.962,Y 28.3672,Z 161,A 11.1206,B 14.087,C -0.0636,E1 14.2438,E2 798.7234} C_DIS
LIN {X 128.9556,Y 23.4314,Z 161,A 9.7974,B 14.0869,C -0.0849,E1 14.2444,E2 799.9458} C_DIS
LIN {X 129.6383,Y 19.3119,Z 161,A 7.6858,B 14.0869,C -0.0704,E1 14.2454,E2 802.0933} C_DIS
LIN {X 130.1732,Y 15.2801,Z 161,A 6.0276,B 14.0869,C -0.069,E1 14.246,E2 803.7393} C_DIS
LIN {X 130.5545,Y 11.5894,Z 161,A 4.3453,B 14.0869,C -0.0622,E1 14.2464,E2 805.4306} C_DIS
LIN {X 130.8246,Y 7.9651,Z 161,A 2.8575,B 14.0869,C -0.0607,E1 14.2467,E2 806.9083} C_DIS
LIN {X 131.0107,Y 3.8393,Z 161,A 1.0422,B 14.087,C -0.055,E1 14.2469,E2 808.7269} C_DIS
LIN {X 131.0679,Y 0.2554,Z 161,A -0.589,B 14.087,C -0.0482,E1 14.2469,E2 810.3676} C_DIS
LIN {X 131.0152,Y -3.6794,Z 161,A -2.1484,B 14.087,C -0.0482,E1 14.2469,E2 811.91} C_DIS
LIN {X 130.8718,Y -7.1712,Z 161,A -3.8245,B 14.087,C -0.0389,E1 14.2466,E2 813.6056} C_DIS
LIN {X 130.5723,Y -11.3792,Z 161,A -5.6237,B 14.087,C -0.0348,E1 14.2462,E2 815.4016} C_DIS
LIN {X 130.1007,Y -15.8877,Z 161,A -7.4498,B 14.087,C -0.0338,E1 14.2456,E2 817.2117} C_DIS
LIN {X 129.6,Y -19.559,Z 161,A -9.5405,B 14.0871,C -0.014,E1 14.2448,E2 819.3602} C_DIS
LIN {X 128.9191,Y -23.6351,Z 161,A -10.8195,B 14.0871,C -0.0254,E1 14.2442,E2 820.579} C_DIS
LIN {X 127.8733,Y -28.7582,Z 161,A -12.9619,B 14.0871,C -0.0232,E1 14.243,E2 822.7072} C_DIS
LIN {X 127.3042,Y -31.1817,Z 161,A -14.1865,B 14.0871,C -0.0156,E1 14.2421,E2 823.9495} C_DIS
LIN {X 125.967,Y -36.2097,Z 161,A -16.3911,B 14.0871,C -0.0112,E1 14.2405,E2 826.1488} C_DIS
LIN {X 125.1602,Y -38.906,Z 161,A -17.6238,B 14.0871,C -0.0075,E1 14.2395,E2 827.3833} C_DIS
LIN {X 124.2035,Y -41.8582,Z 161,A -19.0797,B 14.0871,C -0.0005,E1 14.2382,E2 828.8527} C_DIS
LIN {X 122.0248,Y -47.8381,Z 161,A -21.464,B 14.0871,C -0.0052,E1 14.236,E2 831.1932} C_DIS
LIN {X 120.812,Y -50.8229,Z 161,A -23.1743,B 14.0871,C 0.0084,E1 14.2341,E2 832.9414} C_DIS
LIN {X 119.5024,Y -53.8301,Z 161,A -24.5647,B 14.0871,C 0.0111,E1 14.2326,E2 834.3284} C_DIS
LIN {X 117.8664,Y -57.3273,Z 161,A -26.1993,B 14.0871,C 0.0141,E1 14.2306,E2 835.9589} C_DIS
LIN {X 116.3998,Y -60.2498,Z 161,A -27.649,B 14.0871,C 0.0186,E1 14.2288,E2 837.4128} C_DIS
LIN {X 114.5371,Y -63.7198,Z 161,A -29.4743,B 14.0871,C 0.0265,E1 14.2263,E2 839.2528} C_DIS
LIN {X 112.3683,Y -67.4716,Z 161,A -31.3114,B 14.0871,C 0.0298,E1 14.2237,E2 841.0854} C_DIS
LIN {X 110.3179,Y -70.7734,Z 161,A -33.1839,B 14.0871,C 0.0396,E1 14.2209,E2 842.9806} C_DIS
LIN {X 107.4416,Y -75.0683,Z 161,A -35.2618,B 14.0871,C 0.0397,E1 14.2176,E2 845.0398} C_DIS
LIN {X 104.8784,Y -78.61,Z 161,A -37.3393,B 14.0871,C 0.0497,E1 14.2141,E2 847.1395} C_DIS
LIN {X 99.4432,Y -85.3814,Z 161,A -40.7301,B 14.0871,C 0.0462,E1 14.2082,E2 850.4867} C_DIS
LIN {X 97.1947,Y -87.9324,Z 161,A -43.0124,B 14.0869,C 0.0744,E1 14.2038,E2 852.8652} C_DIS
LIN {X 93.4869,Y -91.8645,Z 161,A -44.5781,B 14.087,C 0.055,E1 14.2009,E2 854.3393} C_DIS
LIN {X 89.7272,Y -95.5406,Z 161,A -46.7493,B 14.087,C 0.056,E1 14.1966,E2 856.498} C_DIS
LIN {X 87.5525,Y -97.5369,Z 161,A -48.693,B 14.087,C 0.079,E1 14.1924,E2 858.5209} C_DIS
LIN {X 84.3417,Y -100.3263,Z 161,A -50.1181,B 14.087,C 0.0694,E1 14.1895,E2 859.8966} C_DIS
LIN {X 80.9678,Y -103.0684,Z 161,A -51.9727,B 14.087,C 0.0718,E1 14.1854,E2 861.7479} C_DIS
LIN {X 77.841,Y -105.4502,Z 161,A -53.7148,B 14.087,C 0.0758,E1 14.1815,E2 863.4947} C_DIS
LIN {X 74.716,Y -107.6867,Z 161,A -55.664,B 14.0869,C 0.0872,E1 14.177,E2 865.4777} C_DIS
LIN {X 71.742,Y -109.6911,Z 161,A -56.9638,B 14.0869,C 0.0817,E1 14.174,E2 866.7475} C_DIS
LIN {X 68.3736,Y -111.8211,Z 161,A -58.61,B 14.0869,C 0.0817,E1 14.1701,E2 868.384} C_DIS
LIN {X 65.1256,Y -113.7435,Z 161,A -60.4048,B 14.0869,C 0.0889,E1 14.1658,E2 870.1977} C_DIS
LIN {X 62.0558,Y -115.4468,Z 161,A -61.8139,B 14.0869,C 0.0875,E1 14.1623,E2 871.5934} C_DIS
LIN {X 58.6299,Y -117.2238,Z 161,A -63.4746,B 14.0869,C 0.0892,E1 14.1582,E2 873.2526} C_DIS
LIN {X 54.8233,Y -119.0497,Z 161,A -65.2515,B 14.0869,C 0.0897,E1 14.1538,E2 875.0229} C_DIS
LIN {X 51.7367,Y -120.4233,Z 161,A -66.7656,B 14.0869,C 0.0928,E1 14.1499,E2 876.5429} C_DIS
LIN {X 48.7603,Y -121.6589,Z 161,A -68.1357,B 14.0869,C 0.0934,E1 14.1463,E2 877.9096} C_DIS
LIN {X 45.1207,Y -123.057,Z 161,A -69.7879,B 14.0869,C 0.0939,E1 14.142,E2 879.5571} C_DIS
LIN {X 42.6902,Y -123.9194,Z 161,A -71.4668,B 14.0867,C 0.1117,E1 14.1374,E2 881.3025} C_DIS
LIN {X 38.6216,Y -125.2472,Z 161,A -72.8311,B 14.0867,C 0.0985,E1 14.1339,E2 882.6082} C_DIS
LIN {X 33.9738,Y -126.5869,Z 161,A -74.9998,B 14.0867,C 0.1021,E1 14.1281,E2 884.785} C_DIS
LIN {X 30.2193,Y -127.5362,Z 161,A -77.06,B 14.0867,C 0.1145,E1 14.1224,E2 886.8902} C_DIS
LIN {X 26.4162,Y -128.3772,Z 161,A -78.4406,B 14.0867,C 0.1062,E1 14.1187,E2 888.2337} C_DIS
LIN {X 22.2685,Y -129.163,Z 161,A -80.1074,B 14.0867,C 0.1022,E1 14.1142,E2 889.8805} C_DIS
LIN {X 19.4805,Y -129.6121,Z 161,A -81.3257,B 14.0867,C 0.1025,E1 14.1108,E2 891.0977} C_DIS
LIN {X 15.1528,Y -130.1884,Z 161,A -83.2872,B 14.0867,C 0.1051,E1 14.1054,E2 893.0668} C_DIS
LIN {X 11.1202,Y -130.5942,Z 161,A -85.0725,B 14.0867,C 0.1062,E1 14.1004,E2 894.8547} C_DIS
LIN {X 6.998,Y -130.8805,Z 161,A -86.941,B 14.0867,C 0.1086,E1 14.0952,E2 896.7316} C_DIS
LIN {X 3.201,Y -131.0285,Z 161,A -88.657,B 14.0867,C 0.1106,E1 14.0903,E2 898.4551} C_DIS
LIN {X 3.201,Y -131.0285,Z 161,A -88.657,B 14.0867,C 0.1106,E1 14.0903,E2 898.4551} C_DIS
Enddeposition()
LIN {X 0.9202,Y -130.1386,Z 161,A -89.2536,B 14.0863,C 0.0905,E1 14.0884,E2 898.9687} C_DIS
Startdeposition()
$VEL.CP = VEL_PRINT
LIN {X 3.2906,Y -130.1014,Z 161,A -87.8055,B 14.0863,C 0.0785,E1 14.0925,E2 897.4719} C_DIS
LIN {X 6.4924,Y -129.9806,Z 161,A -86.461,B 14.0863,C 0.08,E1 14.0963,E2 896.1346} C_DIS
LIN {X 9.6778,Y -129.7824,Z 161,A -85.0637,B 14.0863,C 0.0798,E1 14.1002,E2 894.7374} C_DIS
LIN {X 12.7514,Y -129.5167,Z 161,A -83.7002,B 14.0863,C 0.079,E1 14.104,E2 893.3725} C_DIS
LIN {X 16.6864,Y -129.0685,Z 161,A -82.1472,B 14.0863,C 0.0838,E1 14.1082,E2 891.8412} C_DIS
LIN {X 19.2,Y -128.7204,Z 161,A -80.8708,B 14.0863,C 0.0785,E1 14.1118,E2 890.5451} C_DIS
LIN {X 22.3499,Y -128.2102,Z 161,A -79.4023,B 14.0863,C 0.0757,E1 14.1159,E2 889.068} C_DIS
LIN {X 25.3854,Y -127.6438,Z 161,A -78.0351,B 14.0863,C 0.0745,E1 14.1196,E2 887.699} C_DIS
LIN {X 28.6419,Y -126.9519,Z 161,A -76.6277,B 14.0863,C 0.075,E1 14.1234,E2 886.2974} C_DIS
LIN {X 32.1672,Y -126.1044,Z 161,A -75.1397,B 14.0863,C 0.0769,E1 14.1274,E2 884.8211} C_DIS
LIN {X 34.7719,Y -125.4113,Z 161,A -73.857,B 14.0863,C 0.0729,E1 14.1309,E2 883.526} C_DIS
LIN {X 37.7859,Y -124.5364,Z 161,A -72.4834,B 14.0863,C 0.0718,E1 14.1346,E2 882.1523} C_DIS
LIN {X 40.6927,Y -123.6175,Z 161,A -71.0998,B 14.0864,C 0.0691,E1 14.1383,E2 880.7626} C_DIS
LIN {X 43.8423,Y -122.5355,Z 161,A -69.6797,B 14.0864,C 0.0688,E1 14.142,E2 879.3468} C_DIS
LIN {X 46.9289,Y -121.3867,Z 161,A -68.2366,B 14.0864,C 0.0673,E1 14.1458,E2 877.9032} C_DIS
LIN {X 49.8895,Y -120.2002,Z 161,A -66.8397,B 14.0864,C 0.0657,E1 14.1494,E2 876.5059} C_DIS
LIN {X 53.4619,Y -118.6546,Z 161,A -65.0109,B 14.0864,C 0.0599,E1 14.1541,E2 874.6617} C_DIS
LIN {X 57.0904,Y -116.9527,Z 161,A -63.3842,B 14.0864,C 0.0616,E1 14.1582,E2 873.0499} C_DIS
LIN {X 59.9361,Y -115.5207,Z 161,A -61.9233,B 14.0864,C 0.0577,E1 14.1618,E2 871.5807} C_DIS
LIN {X 62.7444,Y -114.0208,Z 161,A -60.5889,B 14.0864,C 0.0577,E1 14.1651,E2 870.2529} C_DIS
LIN {X 65.5331,Y -112.4412,Z 161,A -59.1806,B 14.0864,C 0.0554,E1 14.1685,E2 868.8436} C_DIS
LIN {X 68.3567,Y -110.7473,Z 161,A -57.6104,B 14.0864,C 0.0492,E1 14.1723,E2 867.2574} C_DIS
LIN {X 71.0497,Y -109.0388,Z 161,A -56.2712,B 14.0864,C 0.0488,E1 14.1754,E2 865.9245} C_DIS
LIN {X 73.7212,Y -107.2505,Z 161,A -54.9436,B 14.0864,C 0.0489,E1 14.1785,E2 864.6059} C_DIS
LIN {X 76.5973,Y -105.2159,Z 161,A -53.4624,B 14.0864,C 0.0482,E1 14.1818,E2 863.1314} C_DIS
LIN {X 79.4709,Y -103.0628,Z 161,A -51.6895,B 14.0865,C 0.0392,E1 14.1858,E2 861.3337} C_DIS
LIN {X 83.1192,Y -100.1434,Z 161,A -49.7724,B 14.0865,C 0.0394,E1 14.1899,E2 859.4311} C_DIS
LIN {X 85.7312,Y -97.9167,Z 161,A -48.1638,B 14.0865,C 0.0333,E1 14.1933,E2 857.8091} C_DIS
LIN {X 88.6065,Y -95.3225,Z 161,A -46.4641,B 14.0865,C 0.0298,E1 14.1968,E2 856.108} C_DIS
LIN {X 91.4694,Y -92.5795,Z 161,A -44.7144,B 14.0865,C 0.0258,E1 14.2003,E2 854.3557} C_DIS
LIN {X 94.7508,Y -89.2176,Z 161,A -42.7915,B 14.0865,C 0.0258,E1 14.204,E2 852.4478} C_DIS
LIN {X 97.4582,Y -86.2518,Z 161,A -41.056,B 14.0865,C 0.0226,E1 14.2073,E2 850.7141} C_DIS
LIN {X 99.6009,Y -83.7684,Z 161,A -39.498,B 14.0865,C 0.0156,E1 14.2101,E2 849.1406} C_DIS
LIN {X 102.5621,Y -80.1162,Z 161,A -37.5661,B 14.0865,C 0.0149,E1 14.2135,E2 847.2228} C_DIS
LIN {X 104.5348,Y -77.5242,Z 161,A -36.1557,B 14.0865,C 0.0121,E1 14.2158,E2 845.8134} C_DIS
LIN {X 106.4012,Y -74.9417,Z 161,A -34.769,B 14.0865,C 0.0091,E1 14.2181,E2 844.4269} C_DIS
LIN {X 108.5176,Y -71.8436,Z 161,A -33.1121,B 14.0865,C 0.0047,E1 14.2207,E2 842.7673} C_DIS
LIN {X 109.9574,Y -69.6195,Z 161,A -31.9567,B 14.0865,C 0.002,E1 14.2224,E2 841.6118} C_DIS
LIN {X 111.6842,Y -66.8143,Z 161,A -30.469,B 14.0865,C -0.003,E1 14.2245,E2 840.1177} C_DIS
LIN {X 113.2869,Y -64.0598,Z 161,A -29.0024,B 14.0865,C -0.0088,E1 14.2266,E2 838.6417} C_DIS
LIN {X 114.8284,Y -61.2542,Z 161,A -27.7421,B 14.0865,C -0.0078,E1 14.2282,E2 837.3975} C_DIS
LIN {X 116.2925,Y -58.425,Z 161,A -26.3606,B 14.0865,C -0.011,E1 14.23,E2 836.0167} C_DIS
LIN {X 117.7089,Y -55.5158,Z 161,A -24.8701,B 14.0865,C -0.017,E1 14.2318,E2 834.5164} C_DIS
LIN {X 118.9724,Y -52.7513,Z 161,A -23.6323,B 14.0865,C -0.0176,E1 14.2332,E2 833.2889} C_DIS
LIN {X 120.2117,Y -49.8619,Z 161,A -22.2664,B 14.0865,C -0.0209,E1 14.2347,E2 831.9234} C_DIS
LIN {X 121.3856,Y -46.9316,Z 161,A -20.8446,B 14.0865,C -0.0259,E1 14.2361,E2 830.496} C_DIS
LIN {X 122.5706,Y -43.7449,Z 161,A -19.4164,B 14.0865,C -0.028,E1 14.2375,E2 829.074} C_DIS
LIN {X 123.5734,Y -40.8253,Z 161,A -18.0617,B 14.0865,C -0.0317,E1 14.2387,E2 827.7181} C_DIS
LIN {X 124.5372,Y -37.7835,Z 161,A -16.6728,B 14.0865,C -0.0353,E1 14.2398,E2 826.3293} C_DIS
LIN {X 125.4321,Y -34.6979,Z 161,A -15.275,B 14.0865,C -0.0389,E1 14.2409,E2 824.9318} C_DIS
LIN {X 126.3774,Y -31.0826,Z 161,A -13.7202,B 14.0865,C -0.0409,E1 14.242,E2 823.3856} C_DIS
LIN {X 126.9781,Y -28.5271,Z 161,A -12.5001,B 14.0865,C -0.0463,E1 14.2427,E2 822.1564} C_DIS
LIN {X 127.7372,Y -24.9096,Z 161,A -11.0146,B 14.0865,C -0.0466,E1 14.2436,E2 820.6857} C_DIS
LIN {X 128.2339,Y -22.2176,Z 161,A -9.713,B 14.0865,C -0.0533,E1 14.2442,E2 819.3712} C_DIS
LIN {X 128.7355,Y -19.0977,Z 161,A -8.2313,B 14.0865,C -0.0603,E1 14.2448,E2 817.8769} C_DIS
LIN {X 129.1656,Y -15.924,Z 161,A -6.8893,B 14.0865,C -0.0624,E1 14.2453,E2 816.5413} C_DIS
LIN {X 129.5166,Y -12.7526,Z 161,A -5.5317,B 14.0865,C -0.0651,E1 14.2457,E2 815.1875} C_DIS
LIN {X 129.7902,Y -9.5709,Z 161,A -4.1479,B 14.0865,C -0.0686,E1 14.246,E2 813.8046} C_DIS
LIN {X 130.0184,Y -5.7221,Z 161,A -2.2558,B 14.0864,C -0.0799,E1 14.2463,E2 811.8874} C_DIS
LIN {X 130.1389,Y -1.0976,Z 161,A -0.6136,B 14.0864,C -0.0734,E1 14.2463,E2 810.2896} C_DIS
LIN {X 130.134,Y 1.5996,Z 161,A 0.7666,B 14.0864,C -0.0831,E1 14.2463,E2 808.8851} C_DIS
LIN {X 130.0547,Y 4.7917,Z 161,A 2.2233,B 14.0864,C -0.089,E1 14.2463,E2 807.4207} C_DIS
LIN {X 129.8914,Y 8.0828,Z 161,A 3.5936,B 14.0863,C -0.0907,E1 14.246,E2 806.0582} C_DIS
LIN {X 129.6535,Y 11.2763,Z 161,A 4.9198,B 14.0863,C -0.0923,E1 14.2457,E2 804.7404} C_DIS
LIN {X 129.3389,Y 14.4497,Z 161,A 6.3109,B 14.0863,C -0.096,E1 14.2453,E2 803.3492} C_DIS
LIN {X 128.9461,Y 17.62,Z 161,A 7.7199,B 14.0863,C -0.1003,E1 14.2448,E2 801.9384} C_DIS
LIN {X 128.4926,Y 20.6704,Z 161,A 9.1278,B 14.0862,C -0.1059,E1 14.2442,E2 800.5231} C_DIS
LIN {X 127.9181,Y 23.9632,Z 161,A 10.4904,B 14.0862,C -0.1067,E1 14.2435,E2 799.1718} C_DIS
LIN {X 127.2946,Y 27.0789,Z 161,A 11.9066,B 14.0862,C -0.1114,E1 14.2427,E2 797.7519} C_DIS
LIN {X 126.5942,Y 30.1832,Z 161,A 13.2916,B 14.0862,C -0.1149,E1 14.2418,E2 796.3674} C_DIS
LIN {X 125.8177,Y 33.2717,Z 161,A 14.8123,B 14.0861,C -0.1227,E1 14.2407,E2 794.8312} C_DIS
LIN {X 124.5115,Y 37.8673,Z 161,A 16.7589,B 14.0861,C -0.1237,E1 14.2392,E2 792.901} C_DIS
LIN {X 123.5479,Y 40.9019,Z 161,A 18.282,B 14.086,C -0.1315,E1 14.2379,E2 791.3622} C_DIS
LIN {X 121.9876,Y 45.3444,Z 161,A 20.2246,B 14.086,C -0.1332,E1 14.2361,E2 789.4331} C_DIS
LIN {X 120.7998,Y 48.4195,Z 161,A 21.6333,B 14.086,C -0.1358,E1 14.2346,E2 788.028} C_DIS
LIN {X 119.3209,Y 51.9578,Z 161,A 23.1845,B 14.086,C -0.1361,E1 14.233,E2 786.4915} C_DIS
LIN {X 118.2283,Y 54.3975,Z 161,A 24.4059,B 14.0859,C -0.1406,E1 14.2315,E2 785.2638} C_DIS
LIN {X 116.9521,Y 57.0915,Z 161,A 25.7657,B 14.0859,C -0.1456,E1 14.2299,E2 783.8974} C_DIS
LIN {X 115.5183,Y 59.9406,Z 161,A 27.2332,B 14.0858,C -0.1513,E1 14.228,E2 782.4212} C_DIS
LIN {X 114.0156,Y 62.7537,Z 161,A 28.5483,B 14.0858,C -0.1521,E1 14.2263,E2 781.1155} C_DIS
LIN {X 112.4442,Y 65.528,Z 161,A 29.9496,B 14.0858,C -0.1556,E1 14.2243,E2 779.7133} C_DIS
LIN {X 110.7428,Y 68.364,Z 161,A 31.5383,B 14.0856,C -0.1634,E1 14.222,E2 778.1079} C_DIS
LIN {X 109.0313,Y 71.0613,Z 161,A 32.8951,B 14.0856,C -0.1653,E1 14.2199,E2 776.7559} C_DIS
LIN {X 107.2543,Y 73.7157,Z 161,A 34.1744,B 14.0856,C -0.1648,E1 14.2179,E2 775.4905} C_DIS
LIN {X 105.4228,Y 76.3119,Z 161,A 35.6826,B 14.0856,C -0.1715,E1 14.2155,E2 773.9686} C_DIS
LIN {X 103.0574,Y 79.478,Z 161,A 37.4308,B 14.0856,C -0.1758,E1 14.2125,E2 772.2183} C_DIS
LIN {X 100.6069,Y 82.5578,Z 161,A 39.1651,B 14.0855,C -0.1798,E1 14.2094,E2 770.4826} C_DIS
LIN {X 97.9842,Y 85.6538,Z 161,A 40.9232,B 14.0855,C -0.1829,E1 14.2062,E2 768.7268} C_DIS
LIN {X 94.8055,Y 89.1596,Z 161,A 42.9806,B 14.0854,C -0.1865,E1 14.2023,E2 766.6713} C_DIS
LIN {X 91.5402,Y 92.5091,Z 161,A 44.9162,B 14.0854,C -0.1869,E1 14.1986,E2 764.7493} C_DIS
LIN {X 88.5751,Y 95.3517,Z 161,A 46.6945,B 14.0854,C -0.1896,E1 14.195,E2 762.9737} C_DIS
LIN {X 85.6137,Y 98.0192,Z 161,A 48.4278,B 14.0853,C -0.1923,E1 14.1913,E2 761.2421} C_DIS
LIN {X 82.5557,Y 100.6086,Z 161,A 50.3271,B 14.0852,C -0.1997,E1 14.1872,E2 759.3263} C_DIS
LIN {X 79.395,Y 103.1217,Z 161,A 52.0996,B 14.0852,C -0.2027,E1 14.1833,E2 757.5538} C_DIS
LIN {X 76.2383,Y 105.4762,Z 161,A 53.6717,B 14.0852,C -0.2008,E1 14.1798,E2 756} C_DIS
Enddeposition()
END
